KUKA KRL program: MyProgram_179().src

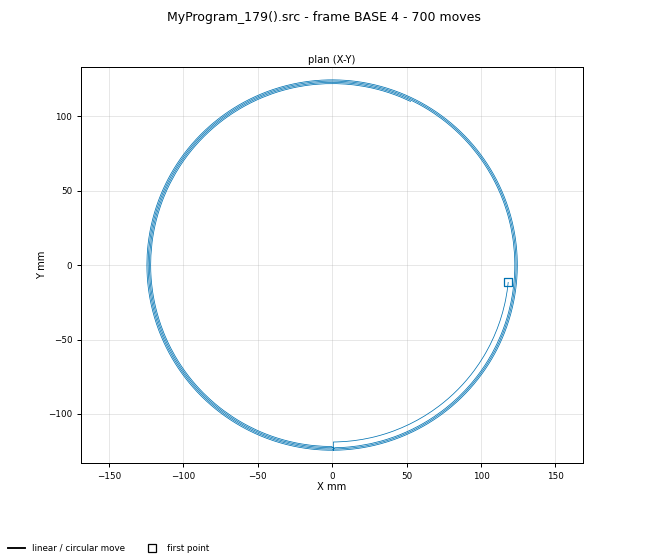
[picture p0: tool path of MyProgram_179().src in frame BASE 4, 700 of 700 moves have a stored position in this frame; points joined in program order, loops and branches not executed]
&ACCESS RVP
&REL 1
&PARAM TEMPLATE = C:\KRC\Roboter\Template\vorgabe
&PARAM EDITMASK = *
DEF MyProgram_179()
; ---- Setting reference (Base) ----
$BASE = BASE_DATA[4]

; --------------------------
; ---- Setting tool (TCP) ----
$TOOL = TOOL_DATA[3]
; --------------------------

$VEL.CP = VEL_APROX_PRINT
Startdeposition()
$VEL.CP = VEL_PRINT
LIN {X 118.2591,Y -11.6542,Z 131,A -9.8058,B 24.9503,C -1.6281,E1 25.1589,E2 455.8963} C_DIS
LIN {X 117.9279,Y -14.6295,Z 131,A -11.2657,B 24.9507,C -1.6226,E1 25.1585,E2 457.3606} C_DIS
LIN {X 117.5311,Y -17.537,Z 131,A -12.6847,B 24.951,C -1.6177,E1 25.1579,E2 458.7826} C_DIS
LIN {X 117.0663,Y -20.4101,Z 131,A -14.029,B 24.951,C -1.616,E1 25.1573,E2 460.1231} C_DIS
LIN {X 116.5481,Y -23.185,Z 131,A -15.4234,B 24.9514,C -1.61,E1 25.1565,E2 461.5236} C_DIS
LIN {X 115.9459,Y -26.0334,Z 131,A -16.854,B 24.9518,C -1.6041,E1 25.1557,E2 462.9597} C_DIS
LIN {X 115.2517,Y -28.9507,Z 131,A -18.2097,B 24.9518,C -1.6038,E1 25.1548,E2 464.3083} C_DIS
LIN {X 114.5261,Y -31.6982,Z 131,A -19.6124,B 24.9522,C -1.5978,E1 25.1538,E2 465.717} C_DIS
LIN {X 113.5377,Y -35.0735,Z 131,A -21.151,B 24.952,C -1.6,E1 25.1526,E2 467.2416} C_DIS
LIN {X 112.7996,Y -37.3815,Z 131,A -22.4561,B 24.9527,C -1.5896,E1 25.1514,E2 468.5637} C_DIS
LIN {X 111.8813,Y -40.0446,Z 131,A -23.8034,B 24.9529,C -1.5859,E1 25.1502,E2 469.9123} C_DIS
LIN {X 110.8682,Y -42.7713,Z 131,A -25.2871,B 24.9534,C -1.5775,E1 25.1487,E2 471.4075} C_DIS
LIN {X 109.7879,Y -45.4717,Z 131,A -26.5696,B 24.9533,C -1.579,E1 25.1473,E2 472.6794} C_DIS
LIN {X 108.6066,Y -48.2246,Z 131,A -27.993,B 24.9535,C -1.5755,E1 25.1458,E2 474.1032} C_DIS
LIN {X 107.4239,Y -50.806,Z 131,A -29.4022,B 24.9539,C -1.5694,E1 25.1441,E2 475.5193} C_DIS
LIN {X 106.142,Y -53.4316,Z 131,A -30.8184,B 24.9541,C -1.5647,E1 25.1423,E2 476.9388} C_DIS
LIN {X 104.7441,Y -56.1219,Z 131,A -32.2269,B 24.9542,C -1.5629,E1 25.1405,E2 478.3442} C_DIS
LIN {X 103.3892,Y -58.5815,Z 131,A -33.6135,B 24.9546,C -1.5573,E1 25.1386,E2 479.7368} C_DIS
LIN {X 101.9208,Y -61.1001,Z 131,A -34.9966,B 24.9547,C -1.5543,E1 25.1366,E2 481.1199} C_DIS
LIN {X 100.3464,Y -63.6522,Z 131,A -36.397,B 24.9549,C -1.5523,E1 25.1346,E2 482.5179} C_DIS
LIN {X 98.8065,Y -66.0182,Z 131,A -37.7837,B 24.9552,C -1.5472,E1 25.1324,E2 483.9098} C_DIS
LIN {X 96.9307,Y -68.7419,Z 131,A -39.2862,B 24.9552,C -1.5472,E1 25.13,E2 485.4051} C_DIS
LIN {X 95.3824,Y -70.8746,Z 131,A -40.7639,B 24.9559,C -1.5336,E1 25.1276,E2 486.9076} C_DIS
LIN {X 93.1999,Y -73.7215,Z 131,A -42.4847,B 24.9562,C -1.5293,E1 25.1246,E2 488.6303} C_DIS
LIN {X 90.4115,Y -77.1157,Z 131,A -44.5876,B 24.9565,C -1.5244,E1 25.1208,E2 490.7352} C_DIS
LIN {X 87.538,Y -80.3628,Z 131,A -46.6704,B 24.9567,C -1.5194,E1 25.1169,E2 492.8205} C_DIS
LIN {X 84.5387,Y -83.5122,Z 131,A -48.7635,B 24.957,C -1.5143,E1 25.1128,E2 494.9166} C_DIS
LIN {X 81.3814,Y -86.5919,Z 131,A -50.8708,B 24.9573,C -1.5101,E1 25.1086,E2 497.0253} C_DIS
LIN {X 78.1228,Y -89.5428,Z 131,A -52.9725,B 24.9575,C -1.506,E1 25.1042,E2 499.1283} C_DIS
LIN {X 74.7881,Y -92.3462,Z 131,A -55.064,B 24.9578,C -1.5016,E1 25.0997,E2 501.222} C_DIS
LIN {X 71.9397,Y -94.582,Z 131,A -56.6673,B 24.9576,C -1.5046,E1 25.0962,E2 502.8124} C_DIS
LIN {X 69.5305,Y -96.3677,Z 131,A -58.1239,B 24.9578,C -1.501,E1 25.0929,E2 504.2723} C_DIS
LIN {X 67.1505,Y -98.0399,Z 131,A -59.4568,B 24.9578,C -1.5015,E1 25.0899,E2 505.5996} C_DIS
LIN {X 64.7475,Y -99.6433,Z 131,A -60.8803,B 24.958,C -1.4972,E1 25.0865,E2 507.0284} C_DIS
LIN {X 62.2378,Y -101.2307,Z 131,A -62.4164,B 24.9584,C -1.4895,E1 25.0829,E2 508.5778} C_DIS
LIN {X 59.7632,Y -102.7102,Z 131,A -63.6661,B 24.9582,C -1.4936,E1 25.0799,E2 509.814} C_DIS
LIN {X 57.2959,Y -104.1069,Z 131,A -65.0773,B 24.9585,C -1.489,E1 25.0764,E2 511.2319} C_DIS
LIN {X 54.1738,Y -105.7643,Z 131,A -66.7164,B 24.9585,C -1.4892,E1 25.0724,E2 512.866} C_DIS
LIN {X 52.0091,Y -106.8461,Z 131,A -67.8926,B 24.9585,C -1.4868,E1 25.0694,E2 514.0448} C_DIS
LIN {X 49.2434,Y -108.1484,Z 131,A -69.339,B 24.9586,C -1.4858,E1 25.0658,E2 515.4899} C_DIS
LIN {X 46.7276,Y -109.2599,Z 131,A -70.7292,B 24.9589,C -1.4807,E1 25.0622,E2 516.8887} C_DIS
LIN {X 44.0427,Y -110.3688,Z 131,A -72.0614,B 24.9589,C -1.4819,E1 25.0588,E2 518.215} C_DIS
LIN {X 41.3309,Y -111.4126,Z 131,A -73.5496,B 24.9592,C -1.4759,E1 25.0548,E2 519.7143} C_DIS
LIN {X 38.6504,Y -112.3713,Z 131,A -74.9079,B 24.9592,C -1.4748,E1 25.0513,E2 521.0724} C_DIS
LIN {X 35.8018,Y -113.3105,Z 131,A -76.4489,B 24.9596,C -1.4686,E1 25.0471,E2 522.6253} C_DIS
LIN {X 32.0327,Y -114.4332,Z 131,A -78.3686,B 24.9598,C -1.4654,E1 25.042,E2 524.5493} C_DIS
LIN {X 28.8636,Y -115.2733,Z 131,A -79.7954,B 24.9595,C -1.4709,E1 25.0382,E2 525.961} C_DIS
LIN {X 26.0318,Y -115.9463,Z 131,A -81.2226,B 24.9596,C -1.4684,E1 25.0343,E2 527.392} C_DIS
LIN {X 23.0081,Y -116.5835,Z 131,A -82.6282,B 24.9595,C -1.471,E1 25.0304,E2 528.7897} C_DIS
LIN {X 20.268,Y -117.0907,Z 131,A -84.0031,B 24.9596,C -1.4685,E1 25.0266,E2 530.1691} C_DIS
LIN {X 17.3202,Y -117.5633,Z 131,A -85.4389,B 24.9596,C -1.4676,E1 25.0227,E2 531.6057} C_DIS
LIN {X 14.4492,Y -117.9503,Z 131,A -86.8237,B 24.9596,C -1.4672,E1 25.0188,E2 532.9902} C_DIS
LIN {X 11.6133,Y -118.2631,Z 131,A -88.2097,B 24.9597,C -1.466,E1 25.015,E2 534.3782} C_DIS
LIN {X 8.7257,Y -118.5119,Z 131,A -89.7515,B 24.9601,C -1.4586,E1 25.0106,E2 535.9366} C_DIS
LIN {X 5.707,Y -118.695,Z 131,A -91.0258,B 24.9597,C -1.4665,E1 25.0071,E2 537.1919} C_DIS
LIN {X 2.9003,Y -118.7965,Z 131,A -92.4392,B 24.9599,C -1.4633,E1 25.0032,E2 538.6124} C_DIS
LIN {X 0.8316,Y -118.8261,Z 131,A -93.3594,B 24.9597,C -1.4666,E1 25.0006,E2 539.5246} C_DIS
Enddeposition()
LIN {X 0.8811,Y -124.3692,Z 132,A -93.1947,B 24.9641,C -1.384,E1 25.0006,E2 539.5559} C_DIS
Startdeposition()
$VEL.CP = VEL_PRINT
LIN {X 5.0073,Y -124.2734,Z 132,A -90.6252,B 24.9624,C -1.417,E1 25.0079,E2 536.9086} C_DIS
LIN {X 9.2445,Y -124.031,Z 132,A -88.5783,B 24.9621,C -1.4223,E1 25.0137,E2 534.8499} C_DIS
LIN {X 13.4703,Y -123.6431,Z 132,A -86.6736,B 24.9621,C -1.421,E1 25.019,E2 532.9497} C_DIS
LIN {X 17.1036,Y -123.1923,Z 132,A -85.0523,B 24.9623,C -1.4189,E1 25.0234,E2 531.3347} C_DIS
LIN {X 20.4851,Y -122.6756,Z 132,A -83.4109,B 24.9621,C -1.4233,E1 25.028,E2 529.6844} C_DIS
LIN {X 24.634,Y -121.9104,Z 132,A -81.626,B 24.9624,C -1.4171,E1 25.0328,E2 527.9163} C_DIS
LIN {X 28.4204,Y -121.0844,Z 132,A -79.6114,B 24.9617,C -1.4301,E1 25.0384,E2 525.8736} C_DIS
LIN {X 32.7722,Y -119.98,Z 132,A -77.5587,B 24.9617,C -1.4316,E1 25.0439,E2 523.8208} C_DIS
LIN {X 37.1507,Y -118.6973,Z 132,A -75.4461,B 24.9614,C -1.4346,E1 25.0496,E2 521.7047} C_DIS
LIN {X 41.4711,Y -117.2578,Z 132,A -73.3668,B 24.9614,C -1.4363,E1 25.0551,E2 519.6253} C_DIS
LIN {X 45.7819,Y -115.6427,Z 132,A -71.268,B 24.9613,C -1.4382,E1 25.0605,E2 517.5267} C_DIS
LIN {X 50.071,Y -113.8509,Z 132,A -69.1721,B 24.9613,C -1.4391,E1 25.0659,E2 515.4336} C_DIS
LIN {X 54.0945,Y -111.9939,Z 132,A -67.217,B 24.9613,C -1.4381,E1 25.0708,E2 513.486} C_DIS
LIN {X 57.1924,Y -110.4452,Z 132,A -65.5312,B 24.9609,C -1.4453,E1 25.0751,E2 511.7878} C_DIS
LIN {X 60.8601,Y -108.4667,Z 132,A -63.6488,B 24.9608,C -1.4469,E1 25.0797,E2 509.9072} C_DIS
LIN {X 64.4363,Y -106.3812,Z 132,A -61.784,B 24.9608,C -1.4483,E1 25.0841,E2 508.0447} C_DIS
LIN {X 67.802,Y -104.2685,Z 132,A -59.9213,B 24.9604,C -1.4535,E1 25.0885,E2 506.1758} C_DIS
LIN {X 71.1094,Y -102.0415,Z 132,A -58.1217,B 24.9604,C -1.4554,E1 25.0927,E2 504.3778} C_DIS
LIN {X 74.3528,Y -99.7029,Z 132,A -56.2324,B 24.96,C -1.4617,E1 25.0969,E2 502.4803} C_DIS
LIN {X 77.768,Y -97.0622,Z 132,A -54.3299,B 24.96,C -1.4617,E1 25.1011,E2 500.5849} C_DIS
LIN {X 80.8617,Y -94.5018,Z 132,A -52.4557,B 24.9597,C -1.4672,E1 25.1051,E2 498.7051} C_DIS
LIN {X 83.8733,Y -91.8379,Z 132,A -50.6415,B 24.9595,C -1.4696,E1 25.1089,E2 496.8924} C_DIS
LIN {X 86.8007,Y -89.0774,Z 132,A -48.733,B 24.9591,C -1.477,E1 25.1127,E2 494.9745} C_DIS
LIN {X 89.8519,Y -85.9986,Z 132,A -46.7528,B 24.9589,C -1.4811,E1 25.1166,E2 492.993} C_DIS
LIN {X 92.7089,Y -82.9096,Z 132,A -44.8836,B 24.9589,C -1.4826,E1 25.1201,E2 491.1286} C_DIS
LIN {X 95.3401,Y -79.8712,Z 132,A -42.9766,B 24.9584,C -1.4903,E1 25.1236,E2 489.212} C_DIS
LIN {X 98.1407,Y -76.4031,Z 132,A -40.938,B 24.9581,C -1.4951,E1 25.1271,E2 487.1716} C_DIS
LIN {X 100.7594,Y -72.915,Z 132,A -38.9836,B 24.958,C -1.4979,E1 25.1303,E2 485.2201} C_DIS
LIN {X 102.9461,Y -69.794,Z 132,A -37.2126,B 24.9576,C -1.5036,E1 25.1331,E2 483.4442} C_DIS
LIN {X 105.1272,Y -66.4622,Z 132,A -35.3917,B 24.9574,C -1.5082,E1 25.1359,E2 481.6216} C_DIS
LIN {X 107.1945,Y -63.0753,Z 132,A -33.5552,B 24.9571,C -1.514,E1 25.1385,E2 479.7809} C_DIS
LIN {X 109.1436,Y -59.6374,Z 132,A -31.82,B 24.957,C -1.515,E1 25.1409,E2 478.0524} C_DIS
LIN {X 110.7562,Y -56.5863,Z 132,A -30.3009,B 24.957,C -1.5162,E1 25.1428,E2 476.5386} C_DIS
LIN {X 112.4871,Y -53.0624,Z 132,A -28.4575,B 24.9565,C -1.5235,E1 25.1451,E2 474.6879} C_DIS
LIN {X 114.0898,Y -49.5222,Z 132,A -26.67,B 24.9562,C -1.5289,E1 25.1471,E2 472.8973} C_DIS
LIN {X 115.6646,Y -45.7259,Z 132,A -24.672,B 24.9556,C -1.5402,E1 25.1492,E2 470.8837} C_DIS
LIN {X 117.2684,Y -41.441,Z 132,A -22.5732,B 24.9552,C -1.5464,E1 25.1512,E2 468.782} C_DIS
LIN {X 118.7069,Y -37.1202,Z 132,A -20.4813,B 24.9548,C -1.5528,E1 25.153,E2 466.6869} C_DIS
LIN {X 119.98,Y -32.7722,Z 132,A -18.4002,B 24.9544,C -1.5592,E1 25.1546,E2 464.6027} C_DIS
LIN {X 121.1136,Y -28.2935,Z 132,A -16.3404,B 24.9543,C -1.5626,E1 25.1559,E2 462.5469} C_DIS
LIN {X 122.0716,Y -23.8197,Z 132,A -14.5054,B 24.9547,C -1.5553,E1 25.157,E2 460.7397} C_DIS
LIN {X 122.6809,Y -20.4536,Z 132,A -12.6743,B 24.9536,C -1.5737,E1 25.1579,E2 458.876} C_DIS
LIN {X 123.3509,Y -15.9277,Z 132,A -10.6309,B 24.9534,C -1.5772,E1 25.1586,E2 456.8363} C_DIS
LIN {X 123.7423,Y -12.5293,Z 132,A -9.0683,B 24.9531,C -1.5817,E1 25.1591,E2 455.2724} C_DIS
LIN {X 124.0398,Y -9.1215,Z 132,A -7.4406,B 24.9527,C -1.5896,E1 25.1595,E2 453.6357} C_DIS
LIN {X 124.2734,Y -5.0073,Z 132,A -5.5644,B 24.9524,C -1.5947,E1 25.1597,E2 451.7588} C_DIS
LIN {X 124.3689,Y -1.0848,Z 132,A -4.0048,B 24.9528,C -1.5878,E1 25.1597,E2 450.2246} C_DIS
LIN {X 124.3535,Y 2.3089,Z 132,A -2.2823,B 24.952,C -1.6011,E1 25.1597,E2 448.4809} C_DIS
LIN {X 124.2254,Y 6.0842,Z 132,A -0.534,B 24.9516,C -1.6073,E1 25.1595,E2 446.7286} C_DIS
LIN {X 123.9906,Y 9.7606,Z 132,A 1.1326,B 24.9514,C -1.6112,E1 25.1592,E2 445.0626} C_DIS
LIN {X 123.6176,Y 13.6985,Z 132,A 2.9082,B 24.9511,C -1.6147,E1 25.1587,E2 443.2893} C_DIS
LIN {X 123.1938,Y 17.093,Z 132,A 4.4717,B 24.9509,C -1.6192,E1 25.1581,E2 441.7245} C_DIS
LIN {X 122.6738,Y 20.4956,Z 132,A 6.1078,B 24.9504,C -1.6268,E1 25.1574,E2 440.0799} C_DIS
LIN {X 121.9104,Y 24.634,Z 132,A 7.8861,B 24.9505,C -1.6247,E1 25.1565,E2 438.317} C_DIS
LIN {X 121.0844,Y 28.4203,Z 132,A 9.8877,B 24.9495,C -1.6415,E1 25.1552,E2 436.2875} C_DIS
LIN {X 119.98,Y 32.7722,Z 132,A 11.9299,B 24.9492,C -1.6466,E1 25.1537,E2 434.2451} C_DIS
LIN {X 118.7005,Y 37.1406,Z 132,A 14.0337,B 24.9488,C -1.6534,E1 25.152,E2 432.1372} C_DIS
LIN {X 117.2542,Y 41.4812,Z 132,A 16.1121,B 24.9485,C -1.6583,E1 25.1501,E2 430.059} C_DIS
LIN {X 115.6427,Y 45.7819,Z 132,A 18.1954,B 24.9482,C -1.6629,E1 25.148,E2 427.9763} C_DIS
LIN {X 113.8956,Y 49.9684,Z 132,A 20.249,B 24.9479,C -1.6672,E1 25.1458,E2 425.9239} C_DIS
LIN {X 112.302,Y 53.453,Z 132,A 21.9196,B 24.9479,C -1.6675,E1 25.1438,E2 424.2617} C_DIS
LIN {X 110.4501,Y 57.183,Z 132,A 23.9271,B 24.9473,C -1.6774,E1 25.1413,E2 422.2413} C_DIS
LIN {X 108.4667,Y 60.8601,Z 132,A 25.7988,B 24.9471,C -1.6801,E1 25.1388,E2 420.3732} C_DIS
LIN {X 106.3812,Y 64.4363,Z 132,A 27.6563,B 24.9469,C -1.6827,E1 25.1361,E2 418.519} C_DIS
LIN {X 104.2685,Y 67.802,Z 132,A 29.4871,B 24.9466,C -1.6876,E1 25.1333,E2 416.6859} C_DIS
LIN {X 102.0415,Y 71.1094,Z 132,A 31.3143,B 24.9464,C -1.6918,E1 25.1305,E2 414.8577} C_DIS
LIN {X 99.7029,Y 74.3528,Z 132,A 33.2055,B 24.9459,C -1.699,E1 25.1273,E2 412.9587} C_DIS
LIN {X 97.0622,Y 77.768,Z 132,A 35.1065,B 24.9459,C -1.6994,E1 25.1241,E2 411.0656} C_DIS
LIN {X 94.5018,Y 80.8617,Z 132,A 36.9807,B 24.9455,C -1.705,E1 25.1207,E2 409.1868} C_DIS
LIN {X 91.8379,Y 83.8733,Z 132,A 38.795,B 24.9454,C -1.7074,E1 25.1173,E2 407.375} C_DIS
LIN {X 89.0774,Y 86.8007,Z 132,A 40.7072,B 24.9449,C -1.7144,E1 25.1136,E2 405.4544} C_DIS
LIN {X 85.9802,Y 89.8694,Z 132,A 42.691,B 24.9447,C -1.7175,E1 25.1096,E2 403.4717} C_DIS
LIN {X 82.9096,Y 92.7088,Z 132,A 44.5914,B 24.9445,C -1.7201,E1 25.1057,E2 401.5726} C_DIS
LIN {X 79.8713,Y 95.3401,Z 132,A 46.4669,B 24.9442,C -1.725,E1 25.1017,E2 399.693} C_DIS
LIN {X 76.4115,Y 98.1342,Z 132,A 48.4659,B 24.9442,C -1.7263,E1 25.0973,E2 397.6982} C_DIS
LIN {X 73.3125,Y 100.47,Z 132,A 50.2018,B 24.9442,C -1.727,E1 25.0934,E2 395.9671} C_DIS
LIN {X 69.9135,Y 102.8649,Z 132,A 52.2086,B 24.9436,C -1.7348,E1 25.0888,E2 393.9487} C_DIS
LIN {X 66.4622,Y 105.1272,Z 132,A 54.0687,B 24.9436,C -1.7358,E1 25.0844,E2 392.0922} C_DIS
LIN {X 63.0753,Y 107.1945,Z 132,A 55.9087,B 24.9433,C -1.7391,E1 25.08,E2 390.2501} C_DIS
LIN {X 59.6374,Y 109.1436,Z 132,A 57.6515,B 24.9433,C -1.7379,E1 25.0758,E2 388.5154} C_DIS
LIN {X 56.5862,Y 110.7562,Z 132,A 59.1717,B 24.9435,C -1.7366,E1 25.072,E2 387.0025} C_DIS
LIN {X 53.0721,Y 112.4825,Z 132,A 61.0234,B 24.9432,C -1.7412,E1 25.0674,E2 385.1447} C_DIS
LIN {X 49.5222,Y 114.0898,Z 132,A 62.8218,B 24.943,C -1.7434,E1 25.0628,E2 383.3455} C_DIS
LIN {X 45.7358,Y 115.6607,Z 132,A 64.8256,B 24.9425,C -1.751,E1 25.0576,E2 381.3282} C_DIS
LIN {X 41.451,Y 117.2648,Z 132,A 66.9383,B 24.9424,C -1.7532,E1 25.052,E2 379.2147} C_DIS
LIN {X 37.11,Y 118.71,Z 132,A 69.0441,B 24.9423,C -1.7548,E1 25.0464,E2 377.109} C_DIS
LIN {X 32.7599,Y 119.9833,Z 132,A 71.1366,B 24.9422,C -1.7565,E1 25.0408,E2 375.0159} C_DIS
LIN {X 28.3039,Y 121.1113,Z 132,A 73.1983,B 24.9422,C -1.755,E1 25.0352,E2 372.9607} C_DIS
LIN {X 23.8302,Y 122.0695,Z 132,A 75.117,B 24.9428,C -1.7469,E1 25.03,E2 371.0637} C_DIS
LIN {X 20.3041,Y 122.7063,Z 132,A 76.9394,B 24.9422,C -1.7558,E1 25.025,E2 369.2222} C_DIS
LIN {X 15.9383,Y 123.3496,Z 132,A 78.9465,B 24.9422,C -1.755,E1 25.0194,E2 367.2186} C_DIS
LIN {X 12.5399,Y 123.7412,Z 132,A 80.5196,B 24.9422,C -1.7551,E1 25.0151,E2 365.6463} C_DIS
LIN {X 9.1108,Y 124.0405,Z 132,A 82.1647,B 24.9421,C -1.7581,E1 25.0105,E2 363.9951} C_DIS
LIN {X 5.0073,Y 124.2734,Z 132,A 84.0495,B 24.9421,C -1.7576,E1 25.0052,E2 362.112} C_DIS
LIN {X 0.8466,Y 124.3717,Z 132,A 85.9248,B 24.9423,C -1.7553,E1 25,E2 360.2424} C_DIS
LIN {X -2.7606,Y 124.3436,Z 132,A 87.6285,B 24.9421,C -1.7569,E1 24.9952,E2 358.5348} C_DIS
LIN {X -6.9449,Y 124.181,Z 132,A 89.5654,B 24.9421,C -1.7566,E1 24.9898,E2 356.5982} C_DIS
LIN {X -11.4331,Y 123.8476,Z 132,A 91.5824,B 24.9424,C -1.7529,E1 24.9842,E2 354.5889} C_DIS
LIN {X -15.446,Y 123.4113,Z 132,A 93.3849,B 24.9427,C -1.7492,E1 24.9792,E2 352.7941} C_DIS
LIN {X -18.8655,Y 122.9351,Z 132,A 94.965,B 24.9427,C -1.7476,E1 24.9749,E2 351.2164} C_DIS
LIN {X -22.6316,Y 122.2987,Z 132,A 96.8269,B 24.9425,C -1.7511,E1 24.9697,E2 349.3444} C_DIS
LIN {X -26.0925,Y 121.6076,Z 132,A 98.5177,B 24.9425,C -1.7527,E1 24.9651,E2 347.6477} C_DIS
LIN {X -30.7627,Y 120.5102,Z 132,A 100.6431,B 24.9428,C -1.7466,E1 24.9594,E2 345.5338} C_DIS
LIN {X -34.9609,Y 119.3594,Z 132,A 102.6898,B 24.9428,C -1.7464,E1 24.9539,E2 343.4844} C_DIS
LIN {X -39.4608,Y 117.9489,Z 132,A 104.8451,B 24.9431,C -1.743,E1 24.9481,E2 341.3333} C_DIS
LIN {X -43.6204,Y 116.4741,Z 132,A 106.9134,B 24.9431,C -1.742,E1 24.9427,E2 339.2633} C_DIS
LIN {X -47.8749,Y 114.7912,Z 132,A 109.058,B 24.9432,C -1.7407,E1 24.9372,E2 337.1169} C_DIS
LIN {X -52.0648,Y 112.9534,Z 132,A 111.1858,B 24.9434,C -1.7384,E1 24.9317,E2 334.9894} C_DIS
LIN {X -55.7249,Y 111.1921,Z 132,A 112.883,B 24.9441,C -1.7274,E1 24.9275,E2 333.314} C_DIS
LIN {X -59.2144,Y 109.375,Z 132,A 114.8019,B 24.944,C -1.7292,E1 24.9228,E2 331.3855} C_DIS
LIN {X -62.6548,Y 107.4398,Z 132,A 116.632,B 24.9441,C -1.7264,E1 24.9184,E2 329.5564} C_DIS
LIN {X -66.119,Y 105.3442,Z 132,A 118.5046,B 24.9443,C -1.7232,E1 24.9139,E2 327.6856} C_DIS
LIN {X -69.3872,Y 103.2199,Z 132,A 120.3097,B 24.9445,C -1.7202,E1 24.9097,E2 325.8819} C_DIS
LIN {X -72.7506,Y 100.8784,Z 132,A 122.2019,B 24.9448,C -1.7165,E1 24.9054,E2 323.992} C_DIS
LIN {X -76.1204,Y 98.3599,Z 132,A 124.1674,B 24.945,C -1.7136,E1 24.901,E2 322.0262} C_DIS
LIN {X -79.2536,Y 95.8536,Z 132,A 126.0049,B 24.9453,C -1.709,E1 24.8971,E2 320.1927} C_DIS
LIN {X -82.3086,Y 93.2432,Z 132,A 127.8871,B 24.9454,C -1.7061,E1 24.8931,E2 318.3099} C_DIS
LIN {X -85.2808,Y 90.5329,Z 132,A 129.7304,B 24.9458,C -1.7013,E1 24.8893,E2 316.4706} C_DIS
LIN {X -88.3499,Y 87.541,Z 132,A 131.739,B 24.946,C -1.698,E1 24.8854,E2 314.4614} C_DIS
LIN {X -91.2936,Y 84.4659,Z 132,A 133.7065,B 24.9463,C -1.6933,E1 24.8816,E2 312.4964} C_DIS
LIN {X -93.9767,Y 81.4702,Z 132,A 135.5492,B 24.9466,C -1.6881,E1 24.8782,E2 310.6579} C_DIS
LIN {X -96.7538,Y 78.1532,Z 132,A 137.6118,B 24.9467,C -1.6859,E1 24.8745,E2 308.5908} C_DIS
LIN {X -99.5188,Y 74.6004,Z 132,A 139.6687,B 24.9471,C -1.6795,E1 24.8711,E2 306.5395} C_DIS
LIN {X -101.865,Y 71.3614,Z 132,A 141.4474,B 24.9476,C -1.6716,E1 24.8682,E2 304.771} C_DIS
LIN {X -104.1279,Y 68.0188,Z 132,A 143.3501,B 24.9479,C -1.6682,E1 24.8653,E2 302.8669} C_DIS
LIN {X -106.2223,Y 64.6974,Z 132,A 145.1951,B 24.9481,C -1.6646,E1 24.8625,E2 301.021} C_DIS
LIN {X -108.2825,Y 61.1879,Z 132,A 147.0318,B 24.9485,C -1.6574,E1 24.86,E2 299.1919} C_DIS
LIN {X -110.0324,Y 57.982,Z 132,A 148.6813,B 24.9489,C -1.6509,E1 24.8578,E2 297.5491} C_DIS
LIN {X -111.4927,Y 55.1227,Z 132,A 150.3193,B 24.9488,C -1.6535,E1 24.8558,E2 295.896} C_DIS
LIN {X -113.2145,Y 51.4919,Z 132,A 152.1403,B 24.9492,C -1.6465,E1 24.8536,E2 294.0817} C_DIS
LIN {X -114.8366,Y 47.7671,Z 132,A 154.0354,B 24.9495,C -1.6418,E1 24.8516,E2 292.1875} C_DIS
LIN {X -116.4853,Y 43.5905,Z 132,A 156.112,B 24.9499,C -1.6357,E1 24.8495,E2 290.1137} C_DIS
LIN {X -118.0029,Y 39.2969,Z 132,A 158.2198,B 24.9502,C -1.6295,E1 24.8476,E2 288.0087} C_DIS
LIN {X -119.3683,Y 34.9302,Z 132,A 160.3319,B 24.9506,C -1.623,E1 24.8459,E2 285.9} C_DIS
LIN {X -120.5668,Y 30.5369,Z 132,A 162.4698,B 24.9509,C -1.618,E1 24.8444,E2 283.7615} C_DIS
LIN {X -121.6143,Y 26.0613,Z 132,A 164.6489,B 24.9512,C -1.6139,E1 24.843,E2 281.5794} C_DIS
LIN {X -122.2987,Y 22.6317,Z 132,A 166.24,B 24.9516,C -1.6077,E1 24.8422,E2 279.9935} C_DIS
LIN {X -123.0368,Y 18.1938,Z 132,A 168.3164,B 24.952,C -1.6011,E1 24.8413,E2 277.9205} C_DIS
LIN {X -123.5818,Y 14.0186,Z 132,A 170.0925,B 24.9528,C -1.5875,E1 24.8407,E2 276.1663} C_DIS
LIN {X -123.9192,Y 10.6306,Z 132,A 171.682,B 24.953,C -1.5833,E1 24.8403,E2 274.5773} C_DIS
LIN {X -124.1865,Y 6.8385,Z 132,A 173.538,B 24.953,C -1.5822,E1 24.84,E2 272.7127} C_DIS
LIN {X -124.3436,Y 2.7606,Z 132,A 175.4043,B 24.9535,C -1.5754,E1 24.8398,E2 270.8513} C_DIS
LIN {X -124.3754,Y 0,Z 132,A 176.8104,B 24.9534,C -1.5772,E1 24.8398,E2 269.4324} C_DIS
LIN {X -124.305,Y -4.1498,Z 132,A 178.6448,B 24.954,C -1.5676,E1 24.8399,E2 267.6101} C_DIS
LIN {X -124.1152,Y -8.0121,Z 132,A -179.616,B 24.9544,C -1.5599,E1 24.8402,E2 265.8787} C_DIS
LIN {X -123.8207,Y -11.7227,Z 132,A -177.8177,B 24.9545,C -1.558,E1 24.8406,E2 264.074} C_DIS
LIN {X -123.4113,Y -15.446,Z 132,A -176.1467,B 24.955,C -1.55,E1 24.8412,E2 262.4121} C_DIS
LIN {X -122.9351,Y -18.8655,Z 132,A -174.5518,B 24.9553,C -1.5451,E1 24.8418,E2 260.8194} C_DIS
LIN {X -122.2987,Y -22.6317,Z 132,A -172.6828,B 24.9553,C -1.5444,E1 24.8427,E2 258.9409} C_DIS
LIN {X -121.6053,Y -26.103,Z 132,A -170.9816,B 24.9554,C -1.5424,E1 24.8437,E2 257.2346} C_DIS
LIN {X -120.5102,Y -30.7627,Z 132,A -168.849,B 24.956,C -1.5323,E1 24.8451,E2 255.1136} C_DIS
LIN {X -119.3624,Y -34.9507,Z 132,A -166.8001,B 24.9562,C -1.5283,E1 24.8467,E2 253.0624} C_DIS
LIN {X -117.9489,Y -39.4608,Z 132,A -164.6259,B 24.9566,C -1.5215,E1 24.8486,E2 250.8919} C_DIS
LIN {X -116.4703,Y -43.6304,Z 132,A -162.5515,B 24.9569,C -1.517,E1 24.8505,E2 248.8164} C_DIS
LIN {X -114.7954,Y -47.8651,Z 132,A -160.4188,B 24.9571,C -1.5124,E1 24.8528,E2 246.6829} C_DIS
LIN {X -112.9579,Y -52.0551,Z 132,A -158.4164,B 24.9578,C -1.5015,E1 24.8551,E2 244.6955} C_DIS
LIN {X -111.4622,Y -55.1849,Z 132,A -156.6941,B 24.9578,C -1.5026,E1 24.8572,E2 242.9612} C_DIS
LIN {X -109.3762,Y -59.2122,Z 132,A -154.6431,B 24.9581,C -1.495,E1 24.8598,E2 240.9173} C_DIS
LIN {X -107.4398,Y -62.6548,Z 132,A -152.8092,B 24.9584,C -1.4907,E1 24.8624,E2 239.0842} C_DIS
LIN {X -105.3499,Y -66.11,Z 132,A -150.9351,B 24.9586,C -1.4863,E1 24.8651,E2 237.2109} C_DIS
LIN {X -103.2199,Y -69.3872,Z 132,A -149.1258,B 24.9589,C -1.4821,E1 24.8679,E2 235.4027} C_DIS
LIN {X -100.8847,Y -72.742,Z 132,A -147.2338,B 24.9591,C -1.4777,E1 24.871,E2 233.5119} C_DIS
LIN {X -98.3599,Y -76.1204,Z 132,A -145.2647,B 24.9593,C -1.4741,E1 24.8743,E2 231.542} C_DIS
LIN {X -95.8536,Y -79.2536,Z 132,A -143.4268,B 24.9596,C -1.4691,E1 24.8775,E2 229.7072} C_DIS
LIN {X -93.2432,Y -82.3086,Z 132,A -141.5442,B 24.9597,C -1.4663,E1 24.881,E2 227.8229} C_DIS
LIN {X -90.5329,Y -85.2808,Z 132,A -139.7018,B 24.96,C -1.4616,E1 24.8845,E2 225.9835} C_DIS
LIN {X -87.5334,Y -88.3573,Z 132,A -137.6918,B 24.9601,C -1.4587,E1 24.8884,E2 223.9719} C_DIS
LIN {X -84.4658,Y -91.2936,Z 132,A -135.7289,B 24.9603,C -1.455,E1 24.8924,E2 222.0097} C_DIS
LIN {X -81.4702,Y -93.9767,Z 132,A -133.8884,B 24.9606,C -1.4507,E1 24.8963,E2 220.1721} C_DIS
LIN {X -78.1532,Y -96.7538,Z 132,A -131.831,B 24.9606,C -1.4499,E1 24.9007,E2 218.1089} C_DIS
LIN {X -74.8466,Y -99.3326,Z 132,A -129.9704,B 24.961,C -1.4431,E1 24.9048,E2 216.2576} C_DIS
LIN {X -71.7638,Y -101.5833,Z 132,A -128.1271,B 24.961,C -1.444,E1 24.9091,E2 214.4058} C_DIS
LIN {X -68.0098,Y -104.1337,Z 132,A -126.102,B 24.9613,C -1.4376,E1 24.9137,E2 212.3894} C_DIS
LIN {X -64.6974,Y -106.2223,Z 132,A -124.3274,B 24.9615,C -1.4334,E1 24.9179,E2 210.619} C_DIS
LIN {X -61.2158,Y -108.2669,Z 132,A -122.4393,B 24.9615,C -1.4321,E1 24.9225,E2 208.7285} C_DIS
LIN {X -57.982,Y -110.0324,Z 132,A -120.7887,B 24.9618,C -1.4276,E1 24.9266,E2 207.084} C_DIS
LIN {X -55.1323,Y -111.488,Z 132,A -119.161,B 24.9615,C -1.433,E1 24.9307,E2 205.4391} C_DIS
LIN {X -51.4919,Y -113.2145,Z 132,A -117.3438,B 24.9617,C -1.429,E1 24.9353,E2 203.627} C_DIS
LIN {X -47.7671,Y -114.8366,Z 132,A -115.461,B 24.9618,C -1.4275,E1 24.9401,E2 201.7433} C_DIS
LIN {X -43.6005,Y -116.4816,Z 132,A -113.3966,B 24.9619,C -1.4256,E1 24.9455,E2 199.6792} C_DIS
LIN {X -39.2868,Y -118.0063,Z 132,A -111.2875,B 24.962,C -1.4238,E1 24.9511,E2 197.5701} C_DIS
LIN {X -34.92,Y -119.3713,Z 132,A -109.1859,B 24.9621,C -1.422,E1 24.9567,E2 195.4693} C_DIS
LIN {X -30.5265,Y -120.5694,Z 132,A -107.0664,B 24.9621,C -1.4218,E1 24.9624,E2 193.3472} C_DIS
LIN {X -26.0717,Y -121.6121,Z 132,A -104.904,B 24.9621,C -1.4233,E1 24.9683,E2 191.1783} C_DIS
LIN {X -22.6316,Y -122.2987,Z 132,A -103.3198,B 24.9621,C -1.4212,E1 24.9726,E2 189.5975} C_DIS
LIN {X -18.2043,Y -123.0352,Z 132,A -101.2598,B 24.9622,C -1.4203,E1 24.9783,E2 187.5379} C_DIS
LIN {X -14.0186,Y -123.5818,Z 132,A -99.4952,B 24.9627,C -1.4112,E1 24.9832,E2 185.7935} C_DIS
LIN {X -10.3674,Y -123.9408,Z 132,A -97.8715,B 24.9629,C -1.4079,E1 24.9877,E2 184.1769} C_DIS
LIN {X -6.7021,Y -124.1936,Z 132,A -96.0457,B 24.9625,C -1.4144,E1 24.9928,E2 182.3351} C_DIS
LIN {X -2.7606,Y -124.3436,Z 132,A -94.1941,B 24.9625,C -1.4163,E1 24.998,E2 180.4786} C_DIS
LIN {X 0.8811,Y -124.3692,Z 132,A -93.1946,B 24.9641,C -1.3838,E1 25.0006,E2 179.5562} C_DIS
Enddeposition()
LIN {X 0.8811,Y -124.3692,Z 132,A -93.1946,B 24.9641,C -1.3838,E1 25.0006,E2 179.5562} C_DIS
Startdeposition()
$VEL.CP = VEL_PRINT
LIN {X 0.1835,Y -123.5364,Z 132,A -93.7224,B 24.9639,C -1.3887,E1 24.9991,E2 180.0724} C_DIS
LIN {X -3.9024,Y -123.474,Z 132,A -95.5701,B 24.9638,C -1.3907,E1 24.994,E2 181.9156} C_DIS
LIN {X -7.765,Y -123.2911,Z 132,A -97.2314,B 24.9635,C -1.3969,E1 24.9894,E2 183.5626} C_DIS
LIN {X -11.607,Y -122.9897,Z 132,A -99.1327,B 24.9637,C -1.3915,E1 24.984,E2 185.4775} C_DIS
LIN {X -15.6673,Y -122.5388,Z 132,A -101.0403,B 24.9637,C -1.3912,E1 24.9787,E2 187.3871} C_DIS
LIN {X -19.6658,Y -121.9607,Z 132,A -102.9178,B 24.9637,C -1.3915,E1 24.9736,E2 189.2654} C_DIS
LIN {X -24.0452,Y -121.1735,Z 132,A -105.0504,B 24.9639,C -1.3891,E1 24.9677,E2 191.4061} C_DIS
LIN {X -28.5026,Y -120.2031,Z 132,A -107.173,B 24.9639,C -1.3898,E1 24.9619,E2 193.5298} C_DIS
LIN {X -33.8934,Y -118.7956,Z 132,A -109.7096,B 24.9636,C -1.3937,E1 24.9551,E2 196.061} C_DIS
LIN {X -37.5713,Y -117.6836,Z 132,A -111.4803,B 24.9636,C -1.3956,E1 24.9504,E2 197.8304} C_DIS
LIN {X -41.5249,Y -116.348,Z 132,A -113.3761,B 24.9633,C -1.399,E1 24.9454,E2 199.7216} C_DIS
LIN {X -44.9979,Y -115.0492,Z 132,A -115.1281,B 24.9633,C -1.3992,E1 24.9408,E2 201.4769} C_DIS
LIN {X -48.7357,Y -113.5156,Z 132,A -116.7313,B 24.9626,C -1.4137,E1 24.9367,E2 203.0493} C_DIS
LIN {X -51.6775,Y -112.2091,Z 132,A -118.5321,B 24.9632,C -1.4011,E1 24.9321,E2 204.8843} C_DIS
LIN {X -55.126,Y -110.5545,Z 132,A -120.4429,B 24.9634,C -1.3971,E1 24.9272,E2 206.8098} C_DIS
LIN {X -59.4263,Y -108.3036,Z 132,A -122.5914,B 24.963,C -1.4048,E1 24.922,E2 208.9459} C_DIS
LIN {X -63.2428,Y -106.1201,Z 132,A -124.6011,B 24.9628,C -1.4091,E1 24.9171,E2 210.9514} C_DIS
LIN {X -65.8635,Y -104.5141,Z 132,A -126.1238,B 24.9629,C -1.4069,E1 24.9135,E2 212.4842} C_DIS
LIN {X -69.7234,Y -101.9796,Z 132,A -128.2134,B 24.9626,C -1.4127,E1 24.9087,E2 214.5668} C_DIS
LIN {X -72.6732,Y -99.8987,Z 132,A -130.1816,B 24.9632,C -1.4023,E1 24.9042,E2 216.5666} C_DIS
LIN {X -75.5303,Y -97.7565,Z 132,A -131.5178,B 24.9622,C -1.4198,E1 24.9013,E2 217.8662} C_DIS
LIN {X -78.8178,Y -95.1259,Z 132,A -133.5087,B 24.9622,C -1.4218,E1 24.897,E2 219.8599} C_DIS
LIN {X -82.087,Y -92.32,Z 132,A -135.5144,B 24.9619,C -1.4254,E1 24.8927,E2 221.8649} C_DIS
LIN {X -85.6751,Y -88.9995,Z 132,A -137.754,B 24.9616,C -1.4314,E1 24.8882,E2 224.0995} C_DIS
LIN {X -88.6369,Y -86.0506,Z 132,A -139.7014,B 24.9614,C -1.4352,E1 24.8844,E2 226.0461} C_DIS
LIN {X -91.5459,Y -82.9496,Z 132,A -141.727,B 24.9614,C -1.4372,E1 24.8805,E2 228.0758} C_DIS
LIN {X -94.4631,Y -79.6109,Z 132,A -143.714,B 24.9609,C -1.4451,E1 24.8769,E2 230.053} C_DIS
LIN {X -96.8075,Y -76.7438,Z 132,A -145.5201,B 24.9609,C -1.4453,E1 24.8738,E2 231.867} C_DIS
LIN {X -99.3239,Y -73.4571,Z 132,A -147.4547,B 24.9606,C -1.4494,E1 24.8705,E2 233.8011} C_DIS
LIN {X -101.7367,Y -70.0773,Z 132,A -149.3405,B 24.9603,C -1.4561,E1 24.8675,E2 235.6802} C_DIS
LIN {X -104.0136,Y -66.6514,Z 132,A -151.3805,B 24.9603,C -1.4553,E1 24.8644,E2 237.7326} C_DIS
LIN {X -106.4899,Y -62.6197,Z 132,A -153.4491,B 24.9597,C -1.4667,E1 24.8614,E2 239.7844} C_DIS
LIN {X -109.7633,Y -56.6866,Z 132,A -156.6913,B 24.9595,C -1.471,E1 24.8571,E2 243.0335} C_DIS
LIN {X -111.6983,Y -52.7698,Z 132,A -158.6525,B 24.959,C -1.4797,E1 24.8547,E2 244.9847} C_DIS
LIN {X -112.9092,Y -50.1264,Z 132,A -160.1977,B 24.9592,C -1.475,E1 24.8529,E2 246.5497} C_DIS
LIN {X -114.8396,Y -45.5327,Z 132,A -162.2865,B 24.9583,C -1.4915,E1 24.8507,E2 248.6107} C_DIS
LIN {X -116.9697,Y -39.7393,Z 132,A -165.3,B 24.9583,C -1.4935,E1 24.8479,E2 251.6366} C_DIS
LIN {X -118.2218,Y -35.8408,Z 132,A -167.1102,B 24.9577,C -1.5032,E1 24.8464,E2 253.434} C_DIS
LIN {X -119.2918,Y -32.1032,Z 132,A -169.0266,B 24.9577,C -1.5038,E1 24.845,E2 255.3601} C_DIS
LIN {X -120.357,Y -27.8449,Z 132,A -171.04,B 24.9572,C -1.5112,E1 24.8436,E2 257.3677} C_DIS
LIN {X -121.2648,Y -23.577,Z 132,A -173.0352,B 24.9568,C -1.5188,E1 24.8425,E2 259.3565} C_DIS
LIN {X -121.9973,Y -19.4341,Z 132,A -175.0078,B 24.9565,C -1.5241,E1 24.8416,E2 261.3281} C_DIS
LIN {X -122.9492,Y -12.0255,Z 132,A -178.6655,B 24.9563,C -1.5269,E1 24.8404,E2 265.0012} C_DIS
LIN {X -123.4007,Y -5.7831,Z 132,A 178.8298,B 24.9548,C -1.5537,E1 24.84,E2 267.457} C_DIS
LIN {X -123.533,Y 0.7267,Z 132,A 175.5614,B 24.9548,C -1.5527,E1 24.8398,E2 270.7475} C_DIS
LIN {X -123.3443,Y 6.8958,Z 132,A 172.5842,B 24.9546,C -1.557,E1 24.8401,E2 273.7323} C_DIS
LIN {X -123.0139,Y 11.3468,Z 132,A 170.5305,B 24.9541,C -1.5645,E1 24.8406,E2 275.7804} C_DIS
LIN {X -122.1665,Y 18.346,Z 132,A 167.2169,B 24.9536,C -1.5733,E1 24.8418,E2 279.0929} C_DIS
LIN {X -121.4682,Y 22.5125,Z 132,A 165.249,B 24.9533,C -1.5793,E1 24.8427,E2 281.0581} C_DIS
LIN {X -120.6929,Y 26.3509,Z 132,A 163.4548,B 24.9529,C -1.5862,E1 24.8438,E2 282.8465} C_DIS
LIN {X -119.7293,Y 30.4307,Z 132,A 161.5476,B 24.9524,C -1.5941,E1 24.845,E2 284.7461} C_DIS
LIN {X -118.7555,Y 34.0334,Z 132,A 159.7519,B 24.9522,C -1.5968,E1 24.8464,E2 286.5457} C_DIS
LIN {X -117.6587,Y 37.6486,Z 132,A 158.0958,B 24.9516,C -1.6066,E1 24.8477,E2 288.188} C_DIS
LIN {X -116.5856,Y 40.8532,Z 132,A 156.34,B 24.9518,C -1.6033,E1 24.8493,E2 289.9616} C_DIS
LIN {X -115.0613,Y 44.967,Z 132,A 154.4171,B 24.9512,C -1.6146,E1 24.8512,E2 291.8685} C_DIS
LIN {X -113.6532,Y 48.4157,Z 132,A 152.6408,B 24.951,C -1.6178,E1 24.8531,E2 293.6469} C_DIS
LIN {X -112.0115,Y 52.1015,Z 132,A 150.7375,B 24.9507,C -1.6222,E1 24.8553,E2 295.5503} C_DIS
LIN {X -110.427,Y 55.3805,Z 132,A 148.8821,B 24.9508,C -1.62,E1 24.8577,E2 297.4208} C_DIS
LIN {X -108.1169,Y 59.7674,Z 132,A 146.7111,B 24.9501,C -1.6324,E1 24.8605,E2 299.5737} C_DIS
LIN {X -106.1231,Y 63.2379,Z 132,A 144.8226,B 24.9498,C -1.6365,E1 24.8632,E2 301.4624} C_DIS
LIN {X -103.8176,Y 66.9558,Z 132,A 142.8508,B 24.9493,C -1.6448,E1 24.8661,E2 303.4244} C_DIS
LIN {X -102.2986,Y 69.2549,Z 132,A 141.3016,B 24.9498,C -1.6366,E1 24.8686,E2 305.0009} C_DIS
LIN {X -99.3298,Y 73.4491,Z 132,A 139.1401,B 24.9488,C -1.6529,E1 24.8721,E2 307.1341} C_DIS
LIN {X -96.8388,Y 76.7041,Z 132,A 137.2086,B 24.9486,C -1.6567,E1 24.8754,E2 309.0657} C_DIS
LIN {X -94.2058,Y 79.9151,Z 132,A 135.3054,B 24.9482,C -1.6628,E1 24.8788,E2 310.9632} C_DIS
LIN {X -91.495,Y 83.0056,Z 132,A 133.3606,B 24.948,C -1.666,E1 24.8824,E2 312.9089} C_DIS
LIN {X -88.7179,Y 85.9669,Z 132,A 131.4672,B 24.9477,C -1.6703,E1 24.886,E2 314.8004} C_DIS
LIN {X -85.7692,Y 88.9088,Z 132,A 129.5097,B 24.9475,C -1.6738,E1 24.8899,E2 316.7576} C_DIS
LIN {X -82.72,Y 91.7535,Z 132,A 127.5363,B 24.9473,C -1.6766,E1 24.894,E2 318.7322} C_DIS
LIN {X -79.3858,Y 94.6531,Z 132,A 125.5067,B 24.947,C -1.6822,E1 24.8983,E2 320.7566} C_DIS
LIN {X -76.0279,Y 97.3706,Z 132,A 123.4917,B 24.9467,C -1.6861,E1 24.9027,E2 322.7699} C_DIS
LIN {X -72.6708,Y 99.9005,Z 132,A 121.5481,B 24.9464,C -1.6905,E1 24.907,E2 324.71} C_DIS
LIN {X -69.2512,Y 102.3011,Z 132,A 119.6084,B 24.9462,C -1.6943,E1 24.9115,E2 326.6471} C_DIS
LIN {X -66.289,Y 104.2447,Z 132,A 117.9197,B 24.9462,C -1.6954,E1 24.9155,E2 328.3385} C_DIS
LIN {X -62.5281,Y 106.5433,Z 132,A 115.9216,B 24.9458,C -1.7013,E1 24.9202,E2 330.3288} C_DIS
LIN {X -59.1913,Y 108.4322,Z 132,A 114.1641,B 24.9455,C -1.7054,E1 24.9245,E2 332.0817} C_DIS
LIN {X -55.9235,Y 110.1522,Z 132,A 112.4237,B 24.9454,C -1.707,E1 24.9288,E2 333.823} C_DIS
LIN {X -52.8743,Y 111.6487,Z 132,A 110.5911,B 24.946,C -1.6979,E1 24.9335,E2 335.6817} C_DIS
LIN {X -49.6022,Y 113.1408,Z 132,A 108.3976,B 24.9473,C -1.6769,E1 24.9393,E2 337.9304} C_DIS
LIN {X -44.4459,Y 115.2628,Z 132,A 106.0613,B 24.9464,C -1.6916,E1 24.9453,E2 340.2368} C_DIS
LIN {X -40.2518,Y 116.7949,Z 132,A 104.458,B 24.9449,C -1.7153,E1 24.9494,E2 341.7869} C_DIS
LIN {X -36.3887,Y 118.0551,Z 132,A 102.5577,B 24.9448,C -1.7168,E1 24.9544,E2 343.6871} C_DIS
LIN {X -32.2977,Y 119.2396,Z 132,A 100.5779,B 24.9446,C -1.7187,E1 24.9597,E2 345.6654} C_DIS
LIN {X -28.8856,Y 120.1112,Z 132,A 98.5546,B 24.9457,C -1.7026,E1 24.9653,E2 347.7299} C_DIS
LIN {X -24.9706,Y 120.9853,Z 132,A 96.971,B 24.9448,C -1.7168,E1 24.9696,E2 349.2816} C_DIS
LIN {X -20.9159,Y 121.7523,Z 132,A 94.6679,B 24.9458,C -1.7005,E1 24.976,E2 351.6257} C_DIS
LIN {X -16.4136,Y 122.4407,Z 132,A 93.1282,B 24.944,C -1.728,E1 24.9801,E2 353.1013} C_DIS
LIN {X -12.4759,Y 122.9053,Z 132,A 91.1628,B 24.9444,C -1.7232,E1 24.9856,E2 355.0793} C_DIS
LIN {X -6.8672,Y 123.3458,Z 132,A 88.5844,B 24.9442,C -1.7257,E1 24.9928,E2 357.6526} C_DIS
LIN {X -2.6822,Y 123.5069,Z 132,A 86.7482,B 24.9438,C -1.7312,E1 24.9978,E2 359.476} C_DIS
LIN {X 0.799,Y 123.5337,Z 132,A 85.2868,B 24.9433,C -1.7387,E1 25.0019,E2 360.9197} C_DIS
LIN {X 3.7135,Y 123.4799,Z 132,A 83.7148,B 24.944,C -1.7286,E1 25.0063,E2 362.5153} C_DIS
LIN {X 8.6027,Y 123.2359,Z 132,A 81.43,B 24.944,C -1.728,E1 25.0127,E2 364.8008} C_DIS
LIN {X 12.9837,Y 122.8518,Z 132,A 79.39,B 24.944,C -1.7277,E1 25.0184,E2 366.8402} C_DIS
LIN {X 17.0151,Y 122.3584,Z 132,A 77.6817,B 24.9436,C -1.7355,E1 25.023,E2 368.5286} C_DIS
LIN {X 21.0913,Y 121.7223,Z 132,A 75.6347,B 24.944,C -1.7286,E1 25.0287,E2 370.5899} C_DIS
LIN {X 24.823,Y 121.0157,Z 132,A 73.8702,B 24.944,C -1.7277,E1 25.0336,E2 372.3545} C_DIS
LIN {X 30.9233,Y 119.6031,Z 132,A 70.9135,B 24.9443,C -1.7235,E1 25.0416,E2 375.3168} C_DIS
LIN {X 35.0851,Y 118.4492,Z 132,A 68.9261,B 24.9443,C -1.7228,E1 25.0469,E2 377.3025} C_DIS
LIN {X 39.1353,Y 117.1737,Z 132,A 66.9256,B 24.9446,C -1.7197,E1 25.0523,E2 379.3066} C_DIS
LIN {X 43.3601,Y 115.6764,Z 132,A 64.8447,B 24.9447,C -1.7177,E1 25.0577,E2 381.3879} C_DIS
LIN {X 46.5568,Y 114.4275,Z 132,A 63.227,B 24.9449,C -1.7148,E1 25.0619,E2 383.0089} C_DIS
LIN {X 50.2944,Y 112.8345,Z 132,A 61.5039,B 24.9445,C -1.7204,E1 25.0663,E2 384.7145} C_DIS
LIN {X 53.0826,Y 111.55,Z 132,A 59.9661,B 24.945,C -1.7132,E1 25.0702,E2 386.2654} C_DIS
LIN {X 56.7697,Y 109.7204,Z 132,A 58.0479,B 24.9452,C -1.7103,E1 25.075,E2 388.1853} C_DIS
LIN {X 60.71,Y 107.5897,Z 132,A 56.025,B 24.9452,C -1.71,E1 25.0799,E2 390.203} C_DIS
LIN {X 64.6485,Y 105.271,Z 132,A 53.906,B 24.9454,C -1.7068,E1 25.085,E2 392.323} C_DIS
LIN {X 67.9483,Y 103.1706,Z 132,A 52.1339,B 24.9454,C -1.7059,E1 25.0891,E2 394.0913} C_DIS
LIN {X 71.2124,Y 100.9461,Z 132,A 50.1864,B 24.946,C -1.6972,E1 25.0936,E2 396.0528} C_DIS
LIN {X 74.895,Y 98.2443,Z 132,A 48.1562,B 24.946,C -1.6977,E1 25.0982,E2 398.0745} C_DIS
LIN {X 78.2239,Y 95.6148,Z 132,A 46.1996,B 24.9462,C -1.6945,E1 25.1024,E2 400.0314} C_DIS
LIN {X 81.3441,Y 92.9751,Z 132,A 44.337,B 24.9463,C -1.6923,E1 25.1064,E2 401.8917} C_DIS
LIN {X 84.199,Y 90.3974,Z 132,A 42.6659,B 24.9463,C -1.6942,E1 25.1098,E2 403.5516} C_DIS
LIN {X 86.9513,Y 87.7543,Z 132,A 40.8108,B 24.9467,C -1.6862,E1 25.1135,E2 405.4179} C_DIS
LIN {X 89.6248,Y 85.021,Z 132,A 39.0475,B 24.9469,C -1.6828,E1 25.1169,E2 407.1817} C_DIS
LIN {X 92.443,Y 81.9481,Z 132,A 37.1775,B 24.947,C -1.6815,E1 25.1204,E2 409.0465} C_DIS
LIN {X 97.2925,Y 76.1274,Z 132,A 33.5846,B 24.9478,C -1.6691,E1 25.1268,E2 412.652} C_DIS
LIN {X 99.7727,Y 72.8463,Z 132,A 31.6892,B 24.9481,C -1.6649,E1 25.13,E2 414.5482} C_DIS
LIN {X 102.2902,Y 69.2674,Z 132,A 29.671,B 24.9483,C -1.6602,E1 25.1332,E2 416.5674} C_DIS
LIN {X 104.5863,Y 65.7492,Z 132,A 27.7556,B 24.9486,C -1.6567,E1 25.136,E2 418.4815} C_DIS
LIN {X 106.5753,Y 62.4732,Z 132,A 26.0488,B 24.9486,C -1.6554,E1 25.1385,E2 420.1826} C_DIS
LIN {X 108.542,Y 58.9907,Z 132,A 24.1674,B 24.949,C -1.649,E1 25.141,E2 422.0694} C_DIS
LIN {X 110.196,Y 55.8369,Z 132,A 22.6999,B 24.9488,C -1.6536,E1 25.1429,E2 423.5183} C_DIS
LIN {X 111.1806,Y 53.8515,Z 132,A 21.0338,B 24.9509,C -1.6187,E1 25.145,E2 425.2576} C_DIS
LIN {X 112.9589,Y 50.0145,Z 132,A 19.6025,B 24.9496,C -1.6395,E1 25.1466,E2 426.6322} C_DIS
LIN {X 114.3531,Y 46.7387,Z 132,A 17.9764,B 24.9499,C -1.6359,E1 25.1483,E2 428.2579} C_DIS
LIN {X 115.6805,Y 43.3494,Z 132,A 16.1479,B 24.9506,C -1.6238,E1 25.1502,E2 430.1047} C_DIS
LIN {X 117.2473,Y 38.9122,Z 132,A 14.0776,B 24.9506,C -1.6228,E1 25.1521,E2 432.1656} C_DIS
LIN {X 118.4621,Y 35.0416,Z 132,A 12.3746,B 24.9505,C -1.626,E1 25.1534,E2 433.8513} C_DIS
LIN {X 119.566,Y 31.0668,Z 132,A 9.6513,B 24.9533,C -1.5794,E1 25.1555,E2 436.6689} C_DIS
LIN {X 120.7421,Y 26.1265,Z 132,A 7.7029,B 24.9525,C -1.5923,E1 25.1566,E2 438.5755} C_DIS
LIN {X 121.8125,Y 20.5608,Z 132,A 5.3183,B 24.9523,C -1.5963,E1 25.1578,E2 440.9369} C_DIS
LIN {X 122.4859,Y 16.077,Z 132,A 3.2791,B 24.9525,C -1.5927,E1 25.1586,E2 442.9724} C_DIS
LIN {X 122.8922,Y 12.6025,Z 132,A 1.6767,B 24.9527,C -1.5885,E1 25.1591,E2 444.5754} C_DIS
LIN {X 123.23,Y 8.6864,Z 132,A -0.1177,B 24.953,C -1.584,E1 25.1595,E2 446.3696} C_DIS
LIN {X 123.4437,Y 4.7626,Z 132,A -2.0075,B 24.9535,C -1.5746,E1 25.1597,E2 448.2703} C_DIS
LIN {X 123.5363,Y 0.2063,Z 132,A -3.978,B 24.9535,C -1.575,E1 25.1597,E2 450.2283} C_DIS
LIN {X 123.4979,Y -3.0777,Z 132,A -5.6431,B 24.9542,C -1.5628,E1 25.1597,E2 451.9122} C_DIS
LIN {X 123.3194,Y -7.3122,Z 132,A -7.6116,B 24.9546,C -1.5562,E1 25.1594,E2 453.8846} C_DIS
LIN {X 122.9992,Y -11.5048,Z 132,A -9.4634,B 24.9547,C -1.5547,E1 25.159,E2 455.7287} C_DIS
LIN {X 122.6449,Y -14.8163,Z 132,A -11.0207,B 24.955,C -1.549,E1 25.1585,E2 457.2903} C_DIS
LIN {X 122.0989,Y -18.7873,Z 132,A -12.8801,B 24.9554,C -1.5429,E1 25.1577,E2 459.1531} C_DIS
LIN {X 121.4028,Y -22.8587,Z 132,A -14.9038,B 24.9561,C -1.5312,E1 25.1567,E2 461.1927} C_DIS
LIN {X 120.4319,Y -27.5173,Z 132,A -16.7629,B 24.9555,C -1.5417,E1 25.1557,E2 463.0161} C_DIS
LIN {X 119.2292,Y -32.3365,Z 132,A -19.2656,B 24.9565,C -1.5241,E1 25.1539,E2 465.5459} C_DIS
LIN {X 117.5793,Y -37.8953,Z 132,A -22.4844,B 24.9585,C -1.4888,E1 25.1512,E2 468.8296} C_DIS
LIN {X 116.041,Y -42.373,Z 132,A -24.0879,B 24.9572,C -1.5117,E1 25.1497,E2 470.3701} C_DIS
LIN {X 114.6016,Y -46.1264,Z 132,A -25.9749,B 24.9576,C -1.5047,E1 25.1478,E2 472.2631} C_DIS
LIN {X 112.5614,Y -50.9008,Z 132,A -28.225,B 24.9576,C -1.5053,E1 25.1453,E2 474.4995} C_DIS
LIN {X 110.9675,Y -54.2892,Z 132,A -30.0737,B 24.9582,C -1.4943,E1 25.1431,E2 476.3642} C_DIS
LIN {X 109.2613,Y -57.647,Z 132,A -31.6118,B 24.9579,C -1.4996,E1 25.1411,E2 477.8817} C_DIS
LIN {X 106.6742,Y -62.3038,Z 132,A -34.2994,B 24.9589,C -1.4813,E1 25.1374,E2 480.5985} C_DIS
LIN {X 104.4843,Y -65.9106,Z 132,A -36.199,B 24.9591,C -1.4785,E1 25.1346,E2 482.4951} C_DIS
LIN {X 102.1245,Y -69.5118,Z 132,A -38.2459,B 24.9595,C -1.4702,E1 25.1314,E2 484.5512} C_DIS
LIN {X 99.5388,Y -73.1668,Z 132,A -40.2529,B 24.9596,C -1.4679,E1 25.1281,E2 486.5539} C_DIS
LIN {X 97.058,Y -76.4259,Z 132,A -42.7351,B 24.9615,C -1.4336,E1 25.1238,E2 489.1055} C_DIS
LIN {X 93.969,Y -80.1942,Z 132,A -44.3926,B 24.9602,C -1.4577,E1 25.1209,E2 490.6985} C_DIS
LIN {X 90.1133,Y -84.5044,Z 132,A -47.0391,B 24.9605,C -1.4525,E1 25.1159,E2 493.3454} C_DIS
LIN {X 85.9874,Y -88.6981,Z 132,A -49.8125,B 24.961,C -1.4435,E1 25.1104,E2 496.1283} C_DIS
LIN {X 82.8483,Y -91.6376,Z 132,A -51.6613,B 24.9608,C -1.446,E1 25.1067,E2 497.9637} C_DIS
LIN {X 79.736,Y -94.3573,Z 132,A -54.1076,B 24.9625,C -1.4153,E1 25.1013,E2 500.4731} C_DIS
LIN {X 76.5299,Y -96.9762,Z 132,A -55.6185,B 24.9616,C -1.4313,E1 25.0981,E2 501.9405} C_DIS
LIN {X 73.2817,Y -99.4541,Z 132,A -57.492,B 24.9618,C -1.4283,E1 25.0939,E2 503.8144} C_DIS
LIN {X 67.6768,Y -103.3498,Z 132,A -60.6643,B 24.9621,C -1.4215,E1 25.0866,E2 506.992} C_DIS
LIN {X 64.0244,Y -105.6507,Z 132,A -62.638,B 24.9623,C -1.4191,E1 25.0819,E2 508.9653} C_DIS
LIN {X 60.3357,Y -107.7996,Z 132,A -64.6093,B 24.9624,C -1.4159,E1 25.0771,E2 510.9382} C_DIS
LIN {X 56.5315,Y -109.8427,Z 132,A -66.6337,B 24.9627,C -1.4113,E1 25.0721,E2 512.9676} C_DIS
LIN {X 53.2451,Y -111.472,Z 132,A -68.3313,B 24.9628,C -1.4087,E1 25.0679,E2 514.6668} C_DIS
LIN {X 49.1467,Y -113.3389,Z 132,A -70.3716,B 24.9628,C -1.4079,E1 25.0627,E2 516.7042} C_DIS
LIN {X 45.1718,Y -114.9813,Z 132,A -72.3921,B 24.9631,C -1.4037,E1 25.0574,E2 518.7298} C_DIS
LIN {X 40.8761,Y -116.5776,Z 132,A -74.2024,B 24.9624,C -1.4163,E1 25.0528,E2 520.5066} C_DIS
LIN {X 37.87,Y -117.5875,Z 132,A -75.7914,B 24.9628,C -1.4087,E1 25.0485,E2 522.1107} C_DIS
LIN {X 34.8417,Y -118.5213,Z 132,A -77.4112,B 24.9633,C -1.3996,E1 25.0441,E2 523.7489} C_DIS
LIN {X 29.5592,Y -119.9471,Z 132,A -79.8912,B 24.9633,C -1.3998,E1 25.0374,E2 526.2248} C_DIS
LIN {X 25.9071,Y -120.7902,Z 132,A -81.7393,B 24.9637,C -1.3928,E1 25.0324,E2 528.087} C_DIS
LIN {X 22.115,Y -121.5404,Z 132,A -83.768,B 24.9643,C -1.38,E1 25.0267,E2 530.1437} C_DIS
LIN {X 18.6562,Y -122.1192,Z 132,A -85.0558,B 24.9635,C -1.3951,E1 25.0233,E2 531.3945} C_DIS
LIN {X 14.0819,Y -122.7307,Z 132,A -87.2257,B 24.9637,C -1.3923,E1 25.0172,E2 533.5694} C_DIS
LIN {X 10.111,Y -123.1209,Z 132,A -88.9883,B 24.9635,C -1.3955,E1 25.0124,E2 535.3232} C_DIS
LIN {X 6.3113,Y -123.3744,Z 132,A -90.6297,B 24.9632,C -1.4007,E1 25.0078,E2 536.9516} C_DIS
LIN {X 3.6437,Y -123.482,Z 132,A -91.9672,B 24.9635,C -1.3956,E1 25.0041,E2 538.301} C_DIS
LIN {X 0.8735,Y -123.5302,Z 132,A -92.8346,B 24.9625,C -1.4153,E1 25.0018,E2 539.1216} C_DIS
Enddeposition()
LIN {X 0.8735,Y -123.5302,Z 132,A -92.8346,B 24.9625,C -1.4153,E1 25.0018,E2 539.1216} C_DIS
Startdeposition()
$VEL.CP = VEL_PRINT
LIN {X 1.8113,Y -122.6845,Z 132,A -91.9403,B 24.9605,C -1.4519,E1 25.0045,E2 538.1406} C_DIS
LIN {X 7.8066,Y -122.4486,Z 132,A -89.3648,B 24.961,C -1.4421,E1 25.0116,E2 535.5892} C_DIS
LIN {X 11.6732,Y -122.1413,Z 132,A -87.4956,B 24.9608,C -1.4458,E1 25.0168,E2 533.7123} C_DIS
LIN {X 17.8044,Y -121.3994,Z 132,A -84.6944,B 24.961,C -1.4436,E1 25.0246,E2 530.9184} C_DIS
LIN {X 25.8157,Y -119.9522,Z 132,A -81.0427,B 24.9612,C -1.4394,E1 25.0346,E2 527.281} C_DIS
LIN {X 33.0586,Y -118.1606,Z 132,A -77.4409,B 24.9607,C -1.4486,E1 25.0444,E2 523.6627} C_DIS
LIN {X 36.7542,Y -117.0643,Z 132,A -75.4792,B 24.9601,C -1.4587,E1 25.0496,E2 521.6807} C_DIS
LIN {X 42.0824,Y -115.2549,Z 132,A -73.1134,B 24.9607,C -1.4492,E1 25.0558,E2 519.342} C_DIS
LIN {X 45.3961,Y -113.9914,Z 132,A -71.228,B 24.9599,C -1.4628,E1 25.0608,E2 517.4286} C_DIS
LIN {X 49.4901,Y -112.2747,Z 132,A -68.6845,B 24.9584,C -1.4894,E1 25.0675,E2 514.8285} C_DIS
LIN {X 53.583,Y -110.3799,Z 132,A -67.3672,B 24.9604,C -1.4535,E1 25.0706,E2 513.5993} C_DIS
LIN {X 57.6917,Y -108.2887,Z 132,A -64.9711,B 24.9596,C -1.4693,E1 25.0766,E2 511.1726} C_DIS
LIN {X 61.3411,Y -106.265,Z 132,A -63.0042,B 24.9593,C -1.4737,E1 25.0814,E2 509.2012} C_DIS
LIN {X 64.8609,Y -104.153,Z 132,A -61.0983,B 24.9591,C -1.4769,E1 25.0859,E2 507.2939} C_DIS
LIN {X 68.21,Y -101.9917,Z 132,A -59.1226,B 24.9586,C -1.4863,E1 25.0905,E2 505.3024} C_DIS
LIN {X 73.6719,Y -98.1189,Z 132,A -56.1031,B 24.9586,C -1.4875,E1 25.0974,E2 502.2907} C_DIS
LIN {X 76.7354,Y -95.7416,Z 132,A -53.6905,B 24.9566,C -1.5219,E1 25.1028,E2 499.8059} C_DIS
LIN {X 80.7038,Y -92.4219,Z 132,A -51.1869,B 24.956,C -1.532,E1 25.1081,E2 497.2883} C_DIS
LIN {X 84.8525,Y -88.6283,Z 132,A -49.5735,B 24.9586,C -1.4871,E1 25.1111,E2 495.7876} C_DIS
LIN {X 89.4888,Y -83.9447,Z 132,A -45.636,B 24.9557,C -1.5384,E1 25.119,E2 491.746} C_DIS
LIN {X 92.8304,Y -80.2327,Z 132,A -44.0939,B 24.9576,C -1.5043,E1 25.1216,E2 490.2912} C_DIS
LIN {X 95.0703,Y -77.5654,Z 132,A -42.255,B 24.9567,C -1.5194,E1 25.1249,E2 488.4252} C_DIS
LIN {X 97.6077,Y -74.3474,Z 132,A -40.4328,B 24.9567,C -1.52,E1 25.1281,E2 486.6102} C_DIS
LIN {X 100.1193,Y -70.9299,Z 132,A -38.4351,B 24.9564,C -1.5264,E1 25.1313,E2 484.6071} C_DIS
LIN {X 102.5024,Y -67.4393,Z 132,A -36.4525,B 24.956,C -1.5325,E1 25.1344,E2 482.62} C_DIS
LIN {X 104.812,Y -63.7903,Z 132,A -34.4663,B 24.9558,C -1.5368,E1 25.1373,E2 480.6337} C_DIS
LIN {X 107.524,Y -59.1047,Z 132,A -31.9596,B 24.9554,C -1.5432,E1 25.1408,E2 478.1249} C_DIS
LIN {X 110.3663,Y -53.6109,Z 132,A -29.2447,B 24.9554,C -1.543,E1 25.1442,E2 475.4248} C_DIS
LIN {X 113.2911,Y -47.1179,Z 132,A -25.827,B 24.9545,C -1.558,E1 25.1481,E2 471.9905} C_DIS
LIN {X 114.7405,Y -43.4658,Z 132,A -23.9776,B 24.9541,C -1.5645,E1 25.15,E2 470.136} C_DIS
LIN {X 116.2597,Y -39.2231,Z 132,A -21.4981,B 24.9526,C -1.5904,E1 25.1522,E2 467.6094} C_DIS
LIN {X 117.4317,Y -35.5578,Z 132,A -20.035,B 24.9533,C -1.579,E1 25.1534,E2 466.1815} C_DIS
LIN {X 118.6251,Y -31.3474,Z 132,A -17.7767,B 24.9522,C -1.5966,E1 25.1551,E2 463.8947} C_DIS
LIN {X 119.4775,Y -27.9279,Z 132,A -16.5218,B 24.9531,C -1.5819,E1 25.1559,E2 462.6817} C_DIS
LIN {X 120.0179,Y -25.5064,Z 132,A -14.7573,B 24.951,C -1.6168,E1 25.1569,E2 460.8453} C_DIS
LIN {X 120.8813,Y -21.035,Z 132,A -13.3395,B 24.9528,C -1.5873,E1 25.1576,E2 459.5052} C_DIS
LIN {X 121.4321,Y -17.5786,Z 132,A -11.2584,B 24.9511,C -1.6155,E1 25.1585,E2 457.3699} C_DIS
LIN {X 121.875,Y -14.1838,Z 132,A -10.0141,B 24.9519,C -1.6026,E1 25.1589,E2 456.1634} C_DIS
LIN {X 122.1726,Y -11.3417,Z 132,A -8.7046,B 24.9517,C -1.6057,E1 25.1592,E2 454.8543} C_DIS
LIN {X 122.4616,Y -7.6025,Z 132,A -6.9217,B 24.9512,C -1.6131,E1 25.1596,E2 453.0646} C_DIS
LIN {X 122.6553,Y -3.2486,Z 132,A -4.7586,B 24.9504,C -1.6263,E1 25.1598,E2 450.8832} C_DIS
LIN {X 122.6948,Y 0.727,Z 132,A -2.8226,B 24.9498,C -1.6365,E1 25.1598,E2 448.9347} C_DIS
LIN {X 122.6108,Y 4.6045,Z 132,A -1.289,B 24.9503,C -1.6282,E1 25.1596,E2 447.4298} C_DIS
LIN {X 122.406,Y 8.4548,Z 132,A 0.7724,B 24.9491,C -1.6474,E1 25.1593,E2 445.3353} C_DIS
LIN {X 121.7639,Y 15.1098,Z 132,A 3.288,B 24.9504,C -1.6266,E1 25.1586,E2 442.8837} C_DIS
LIN {X 121.4111,Y 17.7234,Z 132,A 4.9118,B 24.949,C -1.6505,E1 25.1579,E2 441.2132} C_DIS
LIN {X 120.2124,Y 24.5686,Z 132,A 7.8091,B 24.9494,C -1.6431,E1 25.1565,E2 438.3502} C_DIS
LIN {X 119.717,Y 26.8782,Z 132,A 9.5993,B 24.947,C -1.6816,E1 25.1553,E2 436.4797} C_DIS
LIN {X 118.7753,Y 30.7767,Z 132,A 11.0826,B 24.9479,C -1.6675,E1 25.1543,E2 435.0381} C_DIS
LIN {X 117.8075,Y 34.2935,Z 132,A 12.7624,B 24.9476,C -1.6716,E1 25.153,E2 433.3583} C_DIS
LIN {X 116.4916,Y 38.5274,Z 132,A 14.7736,B 24.9474,C -1.6749,E1 25.1513,E2 431.3507} C_DIS
LIN {X 115.166,Y 42.327,Z 132,A 16.8842,B 24.9463,C -1.6923,E1 25.1493,E2 429.2109} C_DIS
LIN {X 113.2157,Y 47.2971,Z 132,A 19.1935,B 24.9465,C -1.6904,E1 25.1469,E2 426.919} C_DIS
LIN {X 111.0757,Y 52.1245,Z 132,A 21.6959,B 24.9459,C -1.6994,E1 25.144,E2 424.4089} C_DIS
LIN {X 109.2404,Y 55.8686,Z 132,A 23.577,B 24.9457,C -1.7016,E1 25.1416,E2 422.5327} C_DIS
LIN {X 107.2301,Y 59.6365,Z 132,A 25.6945,B 24.945,C -1.7133,E1 25.1388,E2 420.3985} C_DIS
LIN {X 104.3782,Y 64.4983,Z 132,A 28.1656,B 24.945,C -1.7123,E1 25.1353,E2 417.9424} C_DIS
LIN {X 102.2058,Y 67.8881,Z 132,A 30.2712,B 24.944,C -1.7286,E1 25.132,E2 415.809} C_DIS
LIN {X 100.3347,Y 70.6244,Z 132,A 31.5475,B 24.9446,C -1.7189,E1 25.13,E2 414.5617} C_DIS
LIN {X 97.8818,Y 73.9859,Z 132,A 33.5024,B 24.9443,C -1.7244,E1 25.1267,E2 412.6033} C_DIS
LIN {X 93.458,Y 79.501,Z 132,A 36.597,B 24.9444,C -1.722,E1 25.1213,E2 409.5287} C_DIS
LIN {X 91.5185,Y 81.7261,Z 132,A 38.1451,B 24.9437,C -1.7336,E1 25.1184,E2 407.9601} C_DIS
LIN {X 88.6451,Y 84.835,Z 132,A 40.1249,B 24.9434,C -1.7382,E1 25.1146,E2 405.9781} C_DIS
LIN {X 85.719,Y 87.7902,Z 132,A 42.0685,B 24.9431,C -1.7425,E1 25.1107,E2 404.0326} C_DIS
LIN {X 82.8632,Y 90.4903,Z 132,A 43.8741,B 24.9429,C -1.7448,E1 25.1071,E2 402.2287} C_DIS
LIN {X 80.1973,Y 92.861,Z 132,A 45.5473,B 24.9427,C -1.7485,E1 25.1035,E2 400.5535} C_DIS
LIN {X 76.9341,Y 95.5825,Z 132,A 47.5045,B 24.9425,C -1.751,E1 25.0993,E2 398.5978} C_DIS
LIN {X 73.5197,Y 98.2335,Z 132,A 49.5568,B 24.9422,C -1.7563,E1 25.0947,E2 396.5405} C_DIS
LIN {X 68.2301,Y 101.9781,Z 132,A 52.4916,B 24.9422,C -1.757,E1 25.088,E2 393.6142} C_DIS
LIN {X 64.9478,Y 104.099,Z 132,A 54.7121,B 24.9407,C -1.7793,E1 25.0827,E2 391.3481} C_DIS
LIN {X 61.7085,Y 106.0511,Z 132,A 56.0035,B 24.942,C -1.7587,E1 25.0797,E2 390.1093} C_DIS
LIN {X 58.4451,Y 107.8851,Z 132,A 57.9202,B 24.9413,C -1.7693,E1 25.075,E2 388.1731} C_DIS
LIN {X 54.2391,Y 110.0588,Z 132,A 60.403,B 24.9403,C -1.7854,E1 25.0687,E2 385.6588} C_DIS
LIN {X 50.9024,Y 111.641,Z 132,A 61.7977,B 24.9412,C -1.7714,E1 25.0652,E2 384.3008} C_DIS
LIN {X 45.2251,Y 114.0599,Z 132,A 64.7046,B 24.9409,C -1.7757,E1 25.0577,E2 381.3905} C_DIS
LIN {X 41.1778,Y 115.5821,Z 132,A 66.679,B 24.9409,C -1.7755,E1 25.0526,E2 379.4208} C_DIS
LIN {X 37.1394,Y 116.9419,Z 132,A 68.6398,B 24.9409,C -1.7757,E1 25.0474,E2 377.4631} C_DIS
LIN {X 33.2983,Y 118.0935,Z 132,A 70.5073,B 24.9409,C -1.7768,E1 25.0424,E2 375.5962} C_DIS
LIN {X 29.6167,Y 119.0694,Z 132,A 72.4541,B 24.9402,C -1.786,E1 25.037,E2 373.6306} C_DIS
LIN {X 21.2967,Y 120.8357,Z 132,A 75.9678,B 24.9416,C -1.7659,E1 25.0276,E2 370.1687} C_DIS
LIN {X 16.3679,Y 121.6012,Z 132,A 78.475,B 24.9409,C -1.775,E1 25.0206,E2 367.6425} C_DIS
LIN {X 13.0852,Y 121.9982,Z 132,A 80.1233,B 24.9406,C -1.7802,E1 25.016,E2 365.983} C_DIS
LIN {X 8.8552,Y 122.378,Z 132,A 82.5312,B 24.9392,C -1.8004,E1 25.0092,E2 363.5284} C_DIS
LIN {X 4.8809,Y 122.6006,Z 132,A 83.8624,B 24.9409,C -1.7754,E1 25.0056,E2 362.2569} C_DIS
LIN {X -0.0997,Y 122.6986,Z 132,A 86.0726,B 24.9413,C -1.7696,E1 24.9995,E2 360.0607} C_DIS
LIN {X -4.5694,Y 122.6121,Z 132,A 88.7237,B 24.9396,C -1.7954,E1 24.9919,E2 357.3481} C_DIS
LIN {X -8.2158,Y 122.4226,Z 132,A 90.1484,B 24.9405,C -1.7816,E1 24.988,E2 355.9556} C_DIS
LIN {X -14.9298,Y 121.7864,Z 132,A 92.9432,B 24.9417,C -1.7634,E1 24.9804,E2 353.2023} C_DIS
LIN {X -22.9185,Y 120.5383,Z 132,A 97.7729,B 24.9386,C -1.8096,E1 24.9668,E2 348.2584} C_DIS
LIN {X -28.3404,Y 119.3801,Z 132,A 99.5995,B 24.9412,C -1.7718,E1 24.962,E2 346.5193} C_DIS
LIN {X -32.2043,Y 118.3968,Z 132,A 101.5252,B 24.9411,C -1.7728,E1 24.9568,E2 344.5883} C_DIS
LIN {X -36.092,Y 117.2695,Z 132,A 103.4209,B 24.9412,C -1.7709,E1 24.9518,E2 342.6938} C_DIS
LIN {X -40.143,Y 115.9455,Z 132,A 105.4971,B 24.9412,C -1.7724,E1 24.9462,E2 340.6102} C_DIS
LIN {X -45.5358,Y 113.935,Z 132,A 108.2545,B 24.9412,C -1.7719,E1 24.939,E2 337.848} C_DIS
LIN {X -49.6618,Y 112.1984,Z 132,A 110.2232,B 24.9417,C -1.7633,E1 24.934,E2 335.8952} C_DIS
LIN {X -53.7361,Y 110.305,Z 132,A 112.0831,B 24.9427,C -1.7492,E1 24.9294,E2 334.0641} C_DIS
LIN {X -56.0689,Y 109.1379,Z 132,A 113.5315,B 24.9421,C -1.7576,E1 24.9258,E2 332.5919} C_DIS
LIN {X -59.8047,Y 107.1362,Z 132,A 115.4798,B 24.9424,C -1.7527,E1 24.921,E2 330.6495} C_DIS
LIN {X -63.3896,Y 105.055,Z 132,A 117.8604,B 24.9413,C -1.7693,E1 24.9152,E2 328.2222} C_DIS
LIN {X -66.8138,Y 102.9112,Z 132,A 119.3628,B 24.9427,C -1.7483,E1 24.9118,E2 326.7651} C_DIS
LIN {X -70.3167,Y 100.5501,Z 132,A 121.3307,B 24.943,C -1.7441,E1 24.9072,E2 324.8005} C_DIS
LIN {X -73.7649,Y 98.049,Z 132,A 123.334,B 24.9432,C -1.7405,E1 24.9027,E2 322.7985} C_DIS
LIN {X -76.9498,Y 95.5699,Z 132,A 125.2222,B 24.9435,C -1.7365,E1 24.8986,E2 320.9128} C_DIS
LIN {X -80.1942,Y 92.8636,Z 132,A 127.2221,B 24.9437,C -1.7333,E1 24.8944,E2 318.9129} C_DIS
LIN {X -83.3576,Y 90.035,Z 132,A 129.1851,B 24.9441,C -1.7278,E1 24.8903,E2 316.9551} C_DIS
LIN {X -86.4502,Y 87.0708,Z 132,A 131.2017,B 24.9443,C -1.7236,E1 24.8863,E2 314.94} C_DIS
LIN {X -89.4493,Y 83.9868,Z 132,A 133.2207,B 24.9446,C -1.7191,E1 24.8824,E2 312.9231} C_DIS
LIN {X -92.1798,Y 80.9793,Z 132,A 135.1457,B 24.9449,C -1.7155,E1 24.8788,E2 310.998} C_DIS
LIN {X -94.9475,Y 77.716,Z 132,A 137.1308,B 24.9452,C -1.7096,E1 24.8753,E2 309.0178} C_DIS
LIN {X -97.5893,Y 74.3716,Z 132,A 139.1064,B 24.9456,C -1.7036,E1 24.8719,E2 307.0472} C_DIS
LIN {X -100.0267,Y 71.0598,Z 132,A 141.5027,B 24.9446,C -1.7194,E1 24.8679,E2 304.6016} C_DIS
LIN {X -102.3509,Y 67.6687,Z 132,A 142.9091,B 24.9464,C -1.6912,E1 24.8659,E2 303.2554} C_DIS
LIN {X -104.0609,Y 65.0092,Z 132,A 144.4839,B 24.9464,C -1.6912,E1 24.8635,E2 301.6723} C_DIS
LIN {X -106.2594,Y 61.3508,Z 132,A 146.4879,B 24.9467,C -1.6859,E1 24.8606,E2 299.6707} C_DIS
LIN {X -109.6619,Y 55.0361,Z 132,A 149.4561,B 24.9484,C -1.6591,E1 24.8568,E2 296.7505} C_DIS
LIN {X -110.7858,Y 52.7379,Z 132,A 151.0746,B 24.9475,C -1.6741,E1 24.8548,E2 295.0877} C_DIS
LIN {X -112.6294,Y 48.6751,Z 132,A 153.1581,B 24.9479,C -1.6677,E1 24.8524,E2 293.008} C_DIS
LIN {X -114.1498,Y 44.9966,Z 132,A 155.0681,B 24.9481,C -1.6641,E1 24.8504,E2 291.0958} C_DIS
LIN {X -115.7142,Y 40.8068,Z 132,A 157.1773,B 24.9485,C -1.6585,E1 24.8484,E2 288.9881} C_DIS
LIN {X -117.3723,Y 35.7536,Z 132,A 159.2895,B 24.9499,C -1.6343,E1 24.8467,E2 286.9213} C_DIS
LIN {X -118.209,Y 32.8847,Z 132,A 161.026,B 24.9493,C -1.6448,E1 24.8453,E2 285.1499} C_DIS
LIN {X -119.279,Y 28.7603,Z 132,A 163.0298,B 24.9497,C -1.639,E1 24.844,E2 283.1482} C_DIS
LIN {X -120.1097,Y 25.0667,Z 132,A 164.8089,B 24.95,C -1.6337,E1 24.8429,E2 281.3711} C_DIS
LIN {X -120.8515,Y 21.2064,Z 132,A 166.6904,B 24.9502,C -1.6297,E1 24.842,E2 279.488} C_DIS
LIN {X -121.468,Y 17.3258,Z 132,A 168.6967,B 24.9502,C -1.6313,E1 24.8411,E2 277.466} C_DIS
LIN {X -122.3934,Y 8.6346,Z 132,A 172.4442,B 24.9518,C -1.6032,E1 24.8401,E2 273.763} C_DIS
LIN {X -122.6928,Y 1.0416,Z 132,A 175.8763,B 24.9528,C -1.5864,E1 24.8398,E2 270.3503} C_DIS
LIN {X -122.5952,Y -5.0174,Z 132,A 179.0783,B 24.9524,C -1.5934,E1 24.84,E2 267.1123} C_DIS
LIN {X -122.0852,Y -12.2502,Z 132,A -177.071,B 24.9519,C -1.6029,E1 24.8409,E2 263.2158} C_DIS
LIN {X -121.5887,Y -16.4616,Z 132,A -175.7566,B 24.954,C -1.5672,E1 24.8414,E2 261.9787} C_DIS
LIN {X -121.1648,Y -19.3326,Z 132,A -174.1893,B 24.9537,C -1.5722,E1 24.842,E2 260.3902} C_DIS
LIN {X -120.458,Y -23.3343,Z 132,A -172.2845,B 24.954,C -1.5664,E1 24.843,E2 258.4878} C_DIS
LIN {X -119.5775,Y -27.4951,Z 132,A -170.2414,B 24.9542,C -1.5627,E1 24.8442,E2 256.4417} C_DIS
LIN {X -118.5609,Y -31.5901,Z 132,A -168.3176,B 24.9547,C -1.5545,E1 24.8456,E2 254.526} C_DIS
LIN {X -117.4772,Y -35.4083,Z 132,A -166.4382,B 24.955,C -1.55,E1 24.847,E2 252.6467} C_DIS
LIN {X -115.9312,Y -40.1839,Z 132,A -163.2583,B 24.9532,C -1.5801,E1 24.85,E2 249.3768} C_DIS
LIN {X -113.8873,Y -45.6558,Z 132,A -161.5813,B 24.9564,C -1.5251,E1 24.8516,E2 247.8214} C_DIS
LIN {X -112.8354,Y -48.1957,Z 132,A -159.8745,B 24.9556,C -1.5401,E1 24.8535,E2 246.0694} C_DIS
LIN {X -110.9721,Y -52.3449,Z 132,A -157.8704,B 24.9562,C -1.5287,E1 24.8558,E2 244.0817} C_DIS
LIN {X -109.046,Y -56.2484,Z 132,A -154.9173,B 24.9542,C -1.5643,E1 24.8597,E2 241.0278} C_DIS
LIN {X -105.9628,Y -61.8599,Z 132,A -152.9868,B 24.9574,C -1.5085,E1 24.8622,E2 239.2204} C_DIS
LIN {X -104.3045,Y -64.6169,Z 132,A -151.2623,B 24.957,C -1.5144,E1 24.8647,E2 237.473} C_DIS
LIN {X -102.1092,Y -68.0332,Z 132,A -149.4209,B 24.9575,C -1.5069,E1 24.8676,E2 235.64} C_DIS
LIN {X -99.7619,Y -71.4307,Z 132,A -147.4237,B 24.9575,C -1.5051,E1 24.8708,E2 233.6373} C_DIS
LIN {X -97.4812,Y -74.5135,Z 132,A -145.6621,B 24.9579,C -1.4994,E1 24.8737,E2 231.881} C_DIS
LIN {X -94.5548,Y -78.1936,Z 132,A -143.4523,B 24.9581,C -1.4947,E1 24.8776,E2 229.672} C_DIS
LIN {X -91.5691,Y -81.6696,Z 132,A -141.3176,B 24.9584,C -1.4895,E1 24.8815,E2 227.54} C_DIS
LIN {X -88.6845,Y -84.7937,Z 132,A -139.3378,B 24.9587,C -1.4848,E1 24.8853,E2 225.5627} C_DIS
LIN {X -85.9536,Y -87.5599,Z 132,A -137.1275,B 24.9579,C -1.4989,E1 24.8898,E2 223.3095} C_DIS
LIN {X -83.1433,Y -90.2342,Z 132,A -135.6637,B 24.959,C -1.4793,E1 24.8927,E2 221.8865} C_DIS
LIN {X -80.0389,Y -92.9976,Z 132,A -133.7036,B 24.9592,C -1.4763,E1 24.8968,E2 219.9258} C_DIS
LIN {X -76.8105,Y -95.6814,Z 132,A -131.9775,B 24.96,C -1.4619,E1 24.9005,E2 218.2274} C_DIS
LIN {X -74.2685,Y -97.6678,Z 132,A -129.0985,B 24.9566,C -1.5226,E1 24.9073,E2 215.1936} C_DIS
LIN {X -68.1391,Y -102.0389,Z 132,A -126.2534,B 24.9587,C -1.4855,E1 24.9137,E2 212.4274} C_DIS
LIN {X -64.5586,Y -104.3407,Z 132,A -124.6908,B 24.9599,C -1.4627,E1 24.9172,E2 210.914} C_DIS
LIN {X -60.8547,Y -106.5433,Z 132,A -122.6803,B 24.9601,C -1.4597,E1 24.9221,E2 208.9045} C_DIS
LIN {X -57.1195,Y -108.5918,Z 132,A -120.2131,B 24.959,C -1.4793,E1 24.9283,E2 206.3839} C_DIS
LIN {X -53.2059,Y -110.561,Z 132,A -118.831,B 24.9608,C -1.4459,E1 24.9316,E2 205.0777} C_DIS
LIN {X -48.1299,Y -112.8637,Z 132,A -116.3209,B 24.9612,C -1.4386,E1 24.938,E2 202.5789} C_DIS
LIN {X -45.2645,Y -114.0441,Z 132,A -114.5374,B 24.9605,C -1.4528,E1 24.9427,E2 200.7578} C_DIS
LIN {X -41.0859,Y -115.615,Z 132,A -112.477,B 24.9606,C -1.4497,E1 24.9481,E2 198.7004} C_DIS
LIN {X -36.7971,Y -117.0507,Z 132,A -110.364,B 24.9607,C -1.4481,E1 24.9537,E2 196.5873} C_DIS
LIN {X -32.5049,Y -118.3145,Z 132,A -108.124,B 24.9604,C -1.4538,E1 24.9597,E2 194.3302} C_DIS
LIN {X -26.2259,Y -119.8623,Z 132,A -105.2595,B 24.9609,C -1.4449,E1 24.9675,E2 191.4831} C_DIS
LIN {X -20.1486,Y -121.0324,Z 132,A -102.274,B 24.9607,C -1.4483,E1 24.9757,E2 188.4863} C_DIS
LIN {X -15.4623,Y -121.7198,Z 132,A -100.1776,B 24.961,C -1.4424,E1 24.9815,E2 186.4025} C_DIS
LIN {X -11.3917,Y -122.1679,Z 132,A -98.0479,B 24.9605,C -1.4526,E1 24.9875,E2 184.2473} C_DIS
LIN {X -6.3055,Y -122.5355,Z 132,A -95.7254,B 24.9606,C -1.4499,E1 24.9939,E2 181.9306} C_DIS
LIN {X -2.5121,Y -122.6723,Z 132,A -94.0824,B 24.9609,C -1.4439,E1 24.9985,E2 180.3016} C_DIS
LIN {X 0.8683,Y -122.6903,Z 132,A -93.0098,B 24.9622,C -1.4201,E1 25.0013,E2 179.2854} C_DIS
Enddeposition()
LIN {X 0.8683,Y -122.6903,Z 132,A -93.0098,B 24.9622,C -1.4201,E1 25.0013,E2 179.2854} C_DIS
Startdeposition()
$VEL.CP = VEL_PRINT
LIN {X -0.4125,Y -121.8591,Z 132,A -93.9377,B 24.9622,C -1.4192,E1 24.9987,E2 180.2154} C_DIS
LIN {X -6.0514,Y -121.7093,Z 132,A -96.5172,B 24.9622,C -1.4223,E1 24.9915,E2 182.788} C_DIS
LIN {X -11.9551,Y -121.2718,Z 132,A -99.4489,B 24.9625,C -1.4154,E1 24.9833,E2 185.7373} C_DIS
LIN {X -14.9087,Y -120.9444,Z 132,A -101.0613,B 24.963,C -1.4056,E1 24.9788,E2 187.374} C_DIS
LIN {X -20.5782,Y -120.1093,Z 132,A -103.6559,B 24.9627,C -1.411,E1 24.9717,E2 189.958} C_DIS
LIN {X -24.1893,Y -119.4348,Z 132,A -105.881,B 24.9639,C -1.3889,E1 24.9654,E2 192.2382} C_DIS
LIN {X -28.8979,Y -118.3828,Z 132,A -107.5048,B 24.9622,C -1.4196,E1 24.9612,E2 193.7913} C_DIS
LIN {X -32.3384,Y -117.4908,Z 132,A -109.259,B 24.9624,C -1.4168,E1 24.9564,E2 195.5548} C_DIS
LIN {X -36.7369,Y -116.1904,Z 132,A -111.3785,B 24.9622,C -1.4201,E1 24.9508,E2 197.6701} C_DIS
LIN {X -40.3898,Y -114.9719,Z 132,A -113.2554,B 24.9623,C -1.4186,E1 24.9458,E2 199.5542} C_DIS
LIN {X -44.6876,Y -113.3707,Z 132,A -115.3813,B 24.9621,C -1.4221,E1 24.9403,E2 201.6764} C_DIS
LIN {X -47.4092,Y -112.259,Z 132,A -117.1231,B 24.9629,C -1.4072,E1 24.9357,E2 203.4573} C_DIS
LIN {X -50.982,Y -110.6838,Z 132,A -118.5095,B 24.9617,C -1.4296,E1 24.9323,E2 204.794} C_DIS
LIN {X -56.3483,Y -108.0491,Z 132,A -121.402,B 24.9617,C -1.4295,E1 24.9251,E2 207.6944} C_DIS
LIN {X -60.0993,Y -106.0095,Z 132,A -123.456,B 24.9617,C -1.4302,E1 24.92,E2 209.7528} C_DIS
LIN {X -63.5842,Y -103.9563,Z 132,A -125.6154,B 24.9621,C -1.4215,E1 24.9148,E2 211.9395} C_DIS
LIN {X -66.4614,Y -102.1409,Z 132,A -126.9742,B 24.9614,C -1.4348,E1 24.9117,E2 213.271} C_DIS
LIN {X -72.9818,Y -97.589,Z 132,A -130.7214,B 24.9611,C -1.4408,E1 24.9032,E2 217.017} C_DIS
LIN {X -76.0181,Y -95.2422,Z 132,A -132.6354,B 24.9611,C -1.4393,E1 24.8989,E2 218.9417} C_DIS
LIN {X -78.8534,Y -92.9083,Z 132,A -134.2432,B 24.9607,C -1.4479,E1 24.8955,E2 220.5351} C_DIS
LIN {X -82.0108,Y -90.1334,Z 132,A -135.9903,B 24.96,C -1.462,E1 24.8919,E2 222.2555} C_DIS
LIN {X -86.4851,Y -85.8505,Z 132,A -139.1599,B 24.9602,C -1.4567,E1 24.8855,E2 225.4509} C_DIS
LIN {X -89.3475,Y -82.8662,Z 132,A -141.3571,B 24.9606,C -1.45,E1 24.8813,E2 227.6738} C_DIS
LIN {X -91.5373,Y -80.4407,Z 132,A -142.6303,B 24.9598,C -1.4651,E1 24.879,E2 228.9168} C_DIS
LIN {X -94.1532,Y -77.3637,Z 132,A -144.8529,B 24.9603,C -1.4554,E1 24.875,E2 231.1727} C_DIS
LIN {X -96.2944,Y -74.6807,Z 132,A -146.0258,B 24.959,C -1.4786,E1 24.873,E2 232.2958} C_DIS
LIN {X -98.8325,Y -71.2888,Z 132,A -148.1915,B 24.9592,C -1.476,E1 24.8694,E2 234.4783} C_DIS
LIN {X -101.1961,Y -67.8908,Z 132,A -150.0445,B 24.9587,C -1.4851,E1 24.8665,E2 236.3188} C_DIS
LIN {X -103.5491,Y -64.2445,Z 132,A -152.1794,B 24.9587,C -1.4863,E1 24.8633,E2 238.4615} C_DIS
LIN {X -105.4195,Y -61.1279,Z 132,A -154.7002,B 24.9603,C -1.4559,E1 24.8597,E2 241.0678} C_DIS
LIN {X -108.2083,Y -56.0439,Z 132,A -156.7411,B 24.9582,C -1.493,E1 24.8571,E2 243.0313} C_DIS
LIN {X -110.2308,Y -51.952,Z 132,A -158.731,B 24.9575,C -1.5059,E1 24.8547,E2 245.0012} C_DIS
LIN {X -112.041,Y -47.9215,Z 132,A -160.8775,B 24.9573,C -1.5089,E1 24.8523,E2 247.1523} C_DIS
LIN {X -113.1672,Y -45.1993,Z 132,A -162.3569,B 24.9573,C -1.5089,E1 24.8507,E2 248.6399} C_DIS
LIN {X -114.8878,Y -40.6307,Z 132,A -165.0578,B 24.9579,C -1.4984,E1 24.8481,E2 251.3812} C_DIS
LIN {X -116.2007,Y -36.7044,Z 132,A -166.5948,B 24.9566,C -1.5219,E1 24.8468,E2 252.871} C_DIS
LIN {X -117.4557,Y -32.4648,Z 132,A -168.6289,B 24.9561,C -1.5303,E1 24.8453,E2 254.897} C_DIS
LIN {X -118.4353,Y -28.6827,Z 132,A -170.4917,B 24.9559,C -1.5349,E1 24.844,E2 256.7596} C_DIS
LIN {X -119.2733,Y -24.9725,Z 132,A -172.2862,B 24.9556,C -1.5403,E1 24.843,E2 258.5519} C_DIS
LIN {X -119.9948,Y -21.2403,Z 132,A -174.0413,B 24.9551,C -1.5473,E1 24.8421,E2 260.3006} C_DIS
LIN {X -120.5942,Y -17.5165,Z 132,A -175.8301,B 24.9549,C -1.5523,E1 24.8413,E2 262.0881} C_DIS
LIN {X -121.22,Y -12.4753,Z 132,A -178.6561,B 24.9555,C -1.5414,E1 24.8404,E2 264.9571} C_DIS
LIN {X -121.5439,Y -8.7682,Z 132,A 179.9033,B 24.9544,C -1.5602,E1 24.8401,E2 266.3615} C_DIS
LIN {X -121.7915,Y -4.0761,Z 132,A 177.2788,B 24.955,C -1.5498,E1 24.8398,E2 269.0267} C_DIS
LIN {X -121.8605,Y 0.0943,Z 132,A 175.8546,B 24.9533,C -1.579,E1 24.8398,E2 270.3898} C_DIS
LIN {X -121.6864,Y 6.4955,Z 132,A 172.677,B 24.9531,C -1.5817,E1 24.8401,E2 273.58} C_DIS
LIN {X -120.9343,Y 14.9895,Z 132,A 168.6661,B 24.9523,C -1.5948,E1 24.8412,E2 277.5839} C_DIS
LIN {X -120.3857,Y 18.8916,Z 132,A 166.8579,B 24.9519,C -1.6027,E1 24.8419,E2 279.3839} C_DIS
LIN {X -119.714,Y 22.7666,Z 132,A 164.9484,B 24.9517,C -1.6062,E1 24.8429,E2 281.2966} C_DIS
LIN {X -118.9478,Y 26.4813,Z 132,A 163.1844,B 24.9513,C -1.6128,E1 24.8439,E2 283.0552} C_DIS
LIN {X -117.985,Y 30.4846,Z 132,A 161.1976,B 24.951,C -1.6168,E1 24.8452,E2 285.0439} C_DIS
LIN {X -116.8511,Y 34.578,Z 132,A 159.3618,B 24.9502,C -1.6301,E1 24.8466,E2 286.8587} C_DIS
LIN {X -115.1497,Y 39.8796,Z 132,A 156.6174,B 24.95,C -1.633,E1 24.849,E2 289.6119} C_DIS
LIN {X -113.9029,Y 43.3112,Z 132,A 154.8086,B 24.95,C -1.6344,E1 24.8508,E2 291.4275} C_DIS
LIN {X -112.7149,Y 46.3156,Z 132,A 153.1585,B 24.95,C -1.6336,E1 24.8525,E2 293.0888} C_DIS
LIN {X -110.6845,Y 50.9807,Z 132,A 150.8136,B 24.9494,C -1.6429,E1 24.8552,E2 295.4243} C_DIS
LIN {X -108.8968,Y 54.6917,Z 132,A 147.6853,B 24.9521,C -1.5984,E1 24.8594,E2 298.6755} C_DIS
LIN {X -105.1019,Y 61.6721,Z 132,A 145.2943,B 24.948,C -1.6663,E1 24.8624,E2 300.9171} C_DIS
LIN {X -101.9271,Y 66.7893,Z 132,A 141.8472,B 24.9491,C -1.6481,E1 24.8677,E2 304.4252} C_DIS
LIN {X -99.4903,Y 70.3682,Z 132,A 140.2613,B 24.9475,C -1.673,E1 24.8701,E2 305.9595} C_DIS
LIN {X -97.0994,Y 73.6309,Z 132,A 138.352,B 24.9472,C -1.6779,E1 24.8733,E2 307.8663} C_DIS
LIN {X -94.4357,Y 77.0175,Z 132,A 136.3416,B 24.9469,C -1.684,E1 24.8768,E2 309.8716} C_DIS
LIN {X -91.8063,Y 80.1347,Z 132,A 134.3628,B 24.9467,C -1.6863,E1 24.8804,E2 311.8538} C_DIS
LIN {X -88.8981,Y 83.3497,Z 132,A 132.3087,B 24.9464,C -1.6908,E1 24.8843,E2 313.9063} C_DIS
LIN {X -85.9732,Y 86.3625,Z 132,A 130.3613,B 24.946,C -1.6969,E1 24.8881,E2 315.8475} C_DIS
LIN {X -83.0334,Y 89.1922,Z 132,A 128.4522,B 24.9457,C -1.7019,E1 24.8919,E2 317.7526} C_DIS
LIN {X -79.8604,Y 92.0445,Z 132,A 126.4351,B 24.9455,C -1.7061,E1 24.8962,E2 319.7678} C_DIS
LIN {X -76.68,Y 94.7108,Z 132,A 124.435,B 24.9453,C -1.7083,E1 24.9005,E2 321.7702} C_DIS
LIN {X -73.1348,Y 97.4747,Z 132,A 122.3149,B 24.945,C -1.7125,E1 24.9052,E2 323.8879} C_DIS
LIN {X -69.6603,Y 99.9865,Z 132,A 120.317,B 24.9447,C -1.7175,E1 24.9097,E2 325.881} C_DIS
LIN {X -66.7727,Y 101.938,Z 132,A 117.8755,B 24.9467,C -1.6857,E1 24.9156,E2 328.4059} C_DIS
LIN {X -61.8626,Y 104.9904,Z 132,A 115.929,B 24.9443,C -1.7244,E1 24.9201,E2 330.2665} C_DIS
LIN {X -58.1576,Y 107.0869,Z 132,A 113.8784,B 24.9442,C -1.7257,E1 24.9251,E2 332.3198} C_DIS
LIN {X -54.4729,Y 109.0068,Z 132,A 111.9206,B 24.944,C -1.7288,E1 24.9299,E2 334.2756} C_DIS
LIN {X -50.5275,Y 110.8907,Z 132,A 109.9612,B 24.9435,C -1.7363,E1 24.9349,E2 336.2221} C_DIS
LIN {X -46.8866,Y 112.4791,Z 132,A 108.3075,B 24.9427,C -1.7485,E1 24.9391,E2 337.8505} C_DIS
LIN {X -40.529,Y 114.9234,Z 132,A 104.7519,B 24.9435,C -1.737,E1 24.9484,E2 341.4409} C_DIS
LIN {X -36.4608,Y 116.2781,Z 132,A 102.7413,B 24.9433,C -1.7397,E1 24.9538,E2 343.4488} C_DIS
LIN {X -32.4997,Y 117.446,Z 132,A 100.8083,B 24.9431,C -1.7422,E1 24.9589,E2 345.3789} C_DIS
LIN {X -27.7947,Y 118.6482,Z 132,A 98.1386,B 24.9441,C -1.7271,E1 24.9663,E2 348.0882} C_DIS
LIN {X -23.8544,Y 119.5021,Z 132,A 96.8709,B 24.9421,C -1.7569,E1 24.9696,E2 349.2866} C_DIS
LIN {X -17.271,Y 120.6293,Z 132,A 93.6502,B 24.9422,C -1.7555,E1 24.9785,E2 352.5136} C_DIS
LIN {X -11.7973,Y 121.2871,Z 132,A 90.8936,B 24.9426,C -1.7495,E1 24.9862,E2 355.2862} C_DIS
LIN {X -4.3504,Y 121.7814,Z 132,A 87.4451,B 24.9424,C -1.7536,E1 24.9958,E2 358.7261} C_DIS
LIN {X 2.9295,Y 121.8245,Z 132,A 84.2726,B 24.9416,C -1.7657,E1 25.0045,E2 361.8697} C_DIS
LIN {X 9.1081,Y 121.5195,Z 132,A 80.3573,B 24.9446,C -1.7196,E1 25.0157,E2 365.8927} C_DIS
LIN {X 14.5509,Y 120.9886,Z 132,A 78.7485,B 24.9417,C -1.7633,E1 25.0199,E2 367.3968} C_DIS
LIN {X 18.73,Y 120.411,Z 132,A 76.5693,B 24.9424,C -1.7538,E1 25.026,E2 369.5967} C_DIS
LIN {X 21.3542,Y 119.9746,Z 132,A 74.5665,B 24.9447,C -1.7186,E1 25.0318,E2 371.6806} C_DIS
LIN {X 26.6241,Y 118.9155,Z 132,A 72.7681,B 24.9425,C -1.7509,E1 25.0364,E2 373.4001} C_DIS
LIN {X 30.6404,Y 117.9448,Z 132,A 70.8706,B 24.9425,C -1.7519,E1 25.0415,E2 375.2925} C_DIS
LIN {X 34.1622,Y 116.9729,Z 132,A 69.0903,B 24.9428,C -1.7478,E1 25.0463,E2 377.0797} C_DIS
LIN {X 38.4851,Y 115.623,Z 132,A 66.971,B 24.9428,C -1.7465,E1 25.052,E2 379.1979} C_DIS
LIN {X 42.7165,Y 114.1276,Z 132,A 64.9991,B 24.9425,C -1.751,E1 25.0571,E2 381.155} C_DIS
LIN {X 46.3321,Y 112.708,Z 132,A 62.8656,B 24.9436,C -1.7347,E1 25.0627,E2 383.3224} C_DIS
LIN {X 52.6801,Y 109.8837,Z 132,A 59.7887,B 24.9433,C -1.7398,E1 25.0705,E2 386.3794} C_DIS
Enddeposition()
END
